FUNCTION_BLOCK "SysTime"   // FB10, SCL
TITLE = 'Формируем текущее циклическое системное время в MD20 (_TIME)'
{ S7_Optimized_Access := 'FALSE' }
AUTHOR : SAA
FAMILY : xSYSTEM
NAME : SysTime
VERSION : 4.0
// // Особенностью SFC 64 TIME_TCK является выдача времени в [мс]
// // от 0 до 16#7FFFFFFF т.е. необходимо организовать переход
// // от 0 до 16#FFFFFFFF. Побочно вычисляем текущее, максимальное
// // и минимальное время цикла и время работы в [сек]
   VAR_OUTPUT
      Tsek : DInt := 0;   // Текущее время [с]
      Tnow : Time := T#0MS;   // Текущее время цикла [мс]
      Trxm : Real := 0.0;   // Текущее время цикла [с]
      Tmid : Real := 0.0;   // Сглаженное время цикла [с]
      Tmax : Time := T#0MS;   // Максимальное время цикла [мс]
      Tmin : Time := T#24D;   // Минимальное время цикла [мс]
      DTx : Date_And_Time;   // Текущее время PLC
   END_VAR
   VAR
      Tm : Time := T#0MS;   // Сохраненное системное время
      Ts : Time := T#0MS;   // Накопитель для секундного счета
      NSc : Bool := 0;   // Первый проход выполнен
   END_VAR
   VAR_TEMP
      Tx : Time;   // Текущее системное время [мс]
      RV : Int;   // RETVAL
   END_VAR
BEGIN

   // Получаем текущее время PLC
   #RV := RD_LOC_T(OUT => #DTx);
   // Получаем разницу между вызовами TIME_TCK
   #Tx := TIME_TCK();
   #Tnow := T_CONV(INT_TO_DINT(DINT_TO_INT(T_CONV(#Tx - #Tm))));
   #Trxm := DINT_TO_REAL(T_CONV(#Tnow)) * 0.001;
   "_Time_dR" := #Trxm;
   #Tm := #Tx;
   // При перезапуске исключаем ударное изменение времени
   IF ("_ReStart") THEN
       #Tnow := T#0s;
   END_IF;
   // Увеличиваем текущий счетчик системного времени
   "_Time" := "_Time" + #Tnow;
   // Пропускаем первый цикл
   IF (#NSc) THEN
       // Выбираем максимум и минимум цикла
       IF (#NSc & #Tnow > #Tmax) THEN
           #Tmax := #Tnow;
       END_IF;
       IF (#NSc & #Tnow < #Tmin) THEN
           #Tmin := #Tnow;
       END_IF;
       // Сглаженное время цикла [с]
       #Tmid := (#Trxm - #Tmid) * 0.001 + #Tmid;
   END_IF;
   // Получаем время в секундах
   #Ts := #Ts + #Tnow;
   IF (#Ts >= T#1s) THEN
       #Tsek := #Tsek + 1;
       #Ts := #Ts - T#1s;
   END_IF;
   // Устанавливаем флаг выполнения первого прохода
   #NSc := 1;
   // Текущее системное время в "_TIME"
END_FUNCTION_BLOCK

FUNCTION_BLOCK "AiCh_My"   // FB12, SCL
{ S7_Optimized_Access := 'FALSE' }
VERSION : 0.1
   VAR_INPUT
      Yi : Int;   // Текущее значение аналогового входного канала
      Ymax : Int := 27648;   // Значение PIW/PID(Ai/Ad) при 100% входного диапазона
      Ymin : Int;   // Значение PIW/PID(Ai/Ad) при 0% входного диапазона
      Xmax : Real;   // Номинал Px при Ai=100%
      Xmin : Real;   // Номинал Px при Ai=0%
      Ke : Bool;   // Прямое использование канала
      Kf : Real;   // Коэффициент преобразования Ai=>Px (множитель)
      lag_koef : Real := 1.0;   // Множитель для сглаживания колебаний входного сигнала
      PV_AH_Lim : Real;   // Максимальний уровень сигнала
      PV_AL_Lim : Real;   // Минимальный уровень сигнала
      PV_WH_Lim : Real;   // Высокий уровень сигнала
      PV_WL_Lim : Real;   // Низкий уровень сигнала
      EnableAL_Lim : Bool := 1;
   END_VAR
   VAR_OUTPUT
      NDB : UDInt := 0;   // Номер InstanceDB
      Pz : Real;   // Фактическое значение канала
      Px : Real;   // Рабочее значение канала
      AH_LIM : Bool;
      AL_LIM : Bool;
   END_VAR
   VAR
      Alarm_error : Program_Alarm;
      Alarm_AH_Lim : Program_Alarm;
      Alarm_AL_Lim : Program_Alarm;
      Alarm_WH_Lim : Program_Alarm;
      Alarm_WL_Lim : Program_Alarm;
      ME : "DrvME";   // Набор данных для обработки ALARM_D
      initBlock : Bool;
      err : Bool;
   END_VAR
   VAR_TEMP
      Pu : Real;
      TSA : "TANY";   // Структура ANY для определения InstanceDB
      TPA AT TSA : ANY;   // Указатель ANY для определения InstanceDB
   END_VAR
BEGIN
   #err := (#Yi <= -32767 OR #Yi >= 32767);

   IF #Ymax - #Ymin <> 0 AND NOT #err THEN
       IF #Ke THEN
           #Pz := #Yi * #Kf+#Xmin;
       ELSE
           #Pz := ((INT_TO_REAL(#Yi - #Ymin)) / (INT_TO_REAL(#Ymax - #Ymin))) * (#Xmax - #Xmin) + #Xmin;
       END_IF;
      // Сглаживание сигнала
       #Pu := #Pz;
       #Pu := (#Pu - #Px) * #lag_koef + #Px;
       #Px := #Pu;

       IF #Pz < #Xmin THEN
           #Pz := #Xmin;
       END_IF;

       IF #Px < #Xmin THEN
           #Px := #Xmin;
       END_IF;

   ELSE
       IF #Yi <= -32767 THEN
           #Pz := -99.0;
           #Px := -99.0;
       END_IF;

       IF #Yi >= 32767 THEN
           #Pz := 999.0;
           #Px := 999.0;
       END_IF;

       IF #Ymax - #Ymin = 0 THEN
           #Pz := -1.0;
           #Px := -1.0;
       END_IF;
   END_IF;


   // Запрос на инициализацию данных
   IF NOT #initBlock THEN
   // Инициализация данных
       #ME.Pr.N2 := 0;
       #ME.Pr.N3 := 0;
       #ME.Pr.N4 := 0;
       #ME.Pr.N5 := 0;
       #ME.Pr.N6 := 0;
   // Устанавливаем номер данного Instance Data Block
       #TPA := #ME;
       #NDB := #TSA.PTR.DN;
       #initBlock := 1;
   END_IF;


   // Сообщение: Неисправность канала датчика
   #ME.Pr.N1 := #NDB*10;
   #ME.Pr.N4 := #NDB*10;
   #Alarm_error(SIG := #err,
                TIMESTAMP := "TS0",
                SD_1:=#ME.Pr.N1, SD_2 := #ME.Pr.N4);


   // Сообщение: Максимальний уровень
   #AH_LIM := #Px > #PV_AH_Lim AND NOT #err;
   #Alarm_AH_Lim(SIG := #AH_LIM,
                  TIMESTAMP := "TS0",
                  SD_1 := #ME.Pr.N1, SD_2 := #ME.Pr.N4);

    // // Сообщение: Минимальный уровень
    #AL_LIM := #Px < #PV_AL_Lim AND NOT #err;
    #Alarm_AL_Lim(SIG :=#AL_LIM AND #EnableAL_Lim,
                  TIMESTAMP := "TS0",
                  SD_1 := #ME.Pr.N1, SD_2 := #ME.Pr.N4);

    // Сообщение: Высокий уровень
    // #Alarm_WH_Lim(SIG := #Px > #PV_WH_Lim AND NOT #err,
    //               TIMESTAMP := "TS0",
    //               SD_1 := #ME.Pr.N1);

    // Сообщение: Низкий уровень
    // #Alarm_WL_Lim(SIG := #Px < #PV_WL_Lim AND NOT #err,
    //               TIMESTAMP := "TS0",
    //               SD_1 := #ME.Pr.N1);
END_FUNCTION_BLOCK

FUNCTION_BLOCK "FpDW"   // FB18, SCL
{ S7_Optimized_Access := 'FALSE' }
VERSION : 0.1
   VAR
      F : Array[00..95] of Bool;   // Текущее состояние
      D AT F : Array[0..2] of DWord;
      "B" : Array[0..2] of DWord;   // Сохраненное состояние
      Fx : Bool := 0;   // Наличие текущих активных сигналов
      Fp : Bool := 0;   // Импульс при наличии новых сигналов
      Fe : Bool := 0;   // Наличие не сквитированных сигналов
      Fa : Bool := 0;   // Мигающий признак Fe
      Fm : Bool := 0;   // Поиск фронта квитирования
   END_VAR
BEGIN
   // ------------------------------------------------------------------------------------------------------------------------------------------------
   // Квитирование (сброс признака наличия новых сигналов)
   IF (#Fm XOR "_ACK") THEN
       #Fe := #Fe & #Fm;
       #Fm := "_ACK";
   END_IF;
   // ------------------------------------------------------------------------------------------------------------------------------------------------
   // Проверка наличия активных сообщений
   #Fx := (#D[0] OR #D[1] OR #D[2]) <> 0;
   // Проверка наличия новых сообщений
   #Fp := ((#D[0] XOR #"B"[0]) & #D[0] OR (#D[1] XOR #"B"[1]) & #D[1] OR (#D[2] XOR #"B"[2]) & #D[2]) <> 0;
   #Fe := #Fe OR #Fp;
   #Fa := (#Fe & "_Clk08sec") OR (#Fx & NOT #Fe);
   // ------------------------------------------------------------------------------------------------------------------------------------------------
   // Сохранение состояния
   #"B" := #D;
   // Очистка входных данных на время наладки
   // #D[0] := 0;
   // #D[1] := 0;
   // #D[2] := 0;
   // ------------------------------------------------------------------------------------------------------------------------------------------------
END_FUNCTION_BLOCK

FUNCTION_BLOCK "DrvCell"   // FB20, SCL
TITLE = 'Элементарная ячейка управления механизмом (DrvCell)'
{ S7_Optimized_Access := 'FALSE' }
AUTHOR : SAA
FAMILY : xDRIVER
NAME : DrvCell
VERSION : 4.0
// ; S7_blockview := 'small'
   VAR_INPUT
      GRP : UDInt := 0;   // Группа механизмов для HMI
      Chr : DWord := 0;   // Входное слово командного канала
      CFr AT Chr : "DrvCF";
      STr AT Chr : "DrvST";
      Lnr : Bool := 1;   // Наличие связи в линии командного канала
      STu : DWord := 16#1000;   // Дополнительные флаги в слове состояния ST
      SQ1 : Bool := 0;   // Концевой выключатель для Km1
      SQ2 : Bool := 0;   // Концевой выключатель для Km2
      Kx1 : Bool := 0;   // Блок-контакт Km1 (подтверждение срабатывания Km1==Kx1)
      Kx2 : Bool := 0;   // Блок-контакт Km2 (подтверждение срабатывания Km2==Kx2)
      KxA : Bool := 0;   // Блок-контакт Km1&Km2 (совмещенный в механизме)
      KxB : Bool := 0;   // Блок-контакт байпаса (разгон окончен)
      QFx : Bool := 1;   // Питающий автомат цепей механизма (1==включен)
      Flt : Bool := 0;   // Внешняя неисправность (блокирующая) (1==активна по умолчанию)
      Dis : Bool := 0;   // Запрет работы ('Аварийный СТОП' или другой режим) (1==активен)
      Ds1 : Bool := 0;   // Блокировка включения (принудительное отключение) Km1
      Ds2 : Bool := 0;   // Блокировка включения (принудительное отключение) Km2
      DsA : Bool := 0;   // Общая блокировка включения (принудительное отключение) Km1&Km2
      MEn : Bool := 1;   // Разрешение выдачи сообщений для HMI
      Mdx : Bool := 0;   // Режим работы (0==Ручной/1==Автомат)
      Cm1 : Bool := 0;   // Включить Km1 (команда в Mode==1)
      Cm2 : Bool := 0;   // Включить Km2 (команда в Mode==1)
      SB1 : Bool := 0;   // Кнопка включения Km1 (фронт активен) (с фиксацией или без)
      SB2 : Bool := 0;   // Кнопка включения Km2 (фронт активен) (с фиксацией или без)
      OFF : Bool := 0;   // Кнопка 'СТОП' для снятия фиксации (1==активен)
      Ack : Bool := 0;   // Сброс индикации ошибки (квитирование) (1==активен)
      SBe : Bool := 1;   // Разрешение кнопок (при ==0 запрет без отключения)
      SP1 : SInt := 100;   // Уставка задания Km1 (-100..+100)[%] (режим: Ручной)
      SP2 : SInt := -100;   // Уставка задания Km2 (-100..+100)[%] (режим: Ручной)
      SK1 : SInt := 100;   // Уставка задания Km1 (-100..+100)[%] (режим: Автомат)
      SK2 : SInt := -100;   // Уставка задания Km2 (-100..+100)[%] (режим: Автомат)
      Kb_Sb1 : Bool := 0;   // Кнопка SB1 без фиксации (Km1 отключается после отпускания SB1)
      Kb_Sr1 : Bool := 0;   // Кнопка SB1 в режиме переключателя (Вкл/Откл одной кнопкой)
      Kb_Sb2 : Bool := 0;   // Кнопка SB2 без фиксации (Km2 отключается после отпускания SB2)
      Kb_Sr2 : Bool := 0;   // Кнопка SB2 в режиме переключателя (Вкл/Откл одной кнопкой)
      Kb_Ls1 : Bool := 0;   // Индикация Km1 желтым светом (Lr+Lg)
      Kb_Ls2 : Bool := 0;   // Индикация Km2 желтым светом (Lr+Lg)
      Kb_LsA : Bool := 0;   // Используется общая подсветка на оба канала Km1/Km2
      Kb_LsH : Bool := 0;   // Моноцветная импульсная индикация неисправностей
      Kb_HMI : Bool := 0;   // Кнопки в режиме импульса HMI (сброс после использования)
      Ds : DWord := 0;   // Канал системы блокировок
      Nm AT Ds : "DrvNm";
      Md_KxB : Bool := 0;   // KxB выпоняет роль блок-контакта байпаса (разгон окончен)
      Md_SQA : Bool := 0;   // Разрешено наличие обоих SQ одновременно
      Md_RsM : Bool := 0;   // Отключение Km при переходе в ручной режим (Mdx=>0)
      Md_DsE : Bool := 0;   // Разрешено аварийное отключение без выдержки времени
      Md_DsM : Bool := 0;   // Не учитывать блокировку действия как Err+Ds в Mdx==0
      Md_DsA : Bool := 0;   // Не учитывать блокировку действия как Err+Ds в Mdx==1
      Md_RsE : Bool := 0;   // Сброс счетчика отработанного времени по фронту Km1/Km2
      Md_Ack : Bool := 0;   // Сброс сообщений производить по обратному фронту Ack
      Md_Tx1 : Bool := 0;   // Используется отключение Km1 по таймеру Tm1
      Md_Sx1 : Bool := 0;   // Превышение времени работы с Sx1==0 является неисправностью
      Md_Sn1 : Bool := 0;   // Разрешен съезд с SQ1 (Sx1=>0) без команды (при On==0)
      Md_Km1 : Bool := 0;   // Активный сигнал SQ1 отключает Km1 (для удержания установить 0)
      Md_Kx1 : Bool := 0;   // Kx1 выпоняет роль блок-контакта (должен соответствовать Km1)
      Md_Tx2 : Bool := 0;   // Используется отключение Km2 по таймеру Tm2
      Md_Sx2 : Bool := 0;   // Превышение времени работы с Sx2==0 является неисправностью
      Md_Sn2 : Bool := 0;   // Разрешен съезд с SQ2 (Sx2=>0) без команды (при On==0)
      Md_Km2 : Bool := 0;   // Активный сигнал SQ2 отключает Km2 (для удержания установить 0)
      Md_Kx2 : Bool := 0;   // Kx2 выпоняет роль блок-контакта (должен соответствовать Km2)
      Md_Sxx : Bool := 0;   // Необходима проверка SQ2 после отключения Km1
      Md_Tm1 : Time := T#24D;   // Контроль времени работы Km1 (T#0MS/T#24D - без ограничения)
      Md_Tm2 : Time := T#24D;   // Контроль времени работы Km2 (T#0MS/T#24D - без ограничения)
      Md_TmX : Time := T#1S;   // Контроль времени включения Km1&Km2 по БК Kx1&Kx2&KxA
      Md_TmD : Time := T#1S;   // Контроль времени отключения Km1&Km2 по БК Kx1&Kx2&KxA
      Md_TmS : Time := T#0MS;   // Уставка времени разгона после включения KOn
      Md_TmF : Time := T#0MS;   // Уставка времени выбега после отключения KOn
      Md_TmU : Time := T#0MS;   // Уставка времени растормаживания перед пуском Km
      Md_TmL : Time := T#0MS;   // Уставка времени наложения тормоза после отключения KOn
   END_VAR
   VAR_OUTPUT
      NDB : UDInt := 0;   // Номер InstanceDB
      Chx : DWord := 0;   // Исходное слово командного канала
      CFx AT Chx : "DrvCF";
      STx AT Chx : "DrvST";
      Sx1 : Bool := 0;   // Активен SQ1 (Sx1==1)
      Sx2 : Bool := 0;   // Активен SQ2 (Sx2==1)
      Sr1 : Bool := 0;   // Механизм в положении Sx1 (рабочее) и остановлен
      Sr2 : Bool := 0;   // Механизм в положении Sx2 (исходное) и остановлен
      Ks1 : Bool := 0;   // Управление действием Km1 от SB1
      Ks2 : Bool := 0;   // Управление действием Km2 от SB2
      KGo : Bool := 0;   // Наличие активной команды Ks1&Ks2
      KBr : Bool := 0;   // Включение тормоза (растормаживание)
      Km1 : Bool := 0;   // Включен Km1 (контактор замкнут с перекрытием)
      Km2 : Bool := 0;   // Включен Km2 (контактор замкнут с перекрытием)
      KOn : Bool := 0;   // Включено (контакторы замкнуты с перекрытием)
      Run : Bool := 0;   // Разгон закончен (стабильный участок)
      Lg1 : Bool := 0;   // Индикация действия от SB1 (зеленый)
      Lg2 : Bool := 0;   // Индикация действия от SB2 (зеленый)
      Lr1 : Bool := 0;   // Индикация действия от SB1 (красный)
      Lr2 : Bool := 0;   // Индикация действия от SB2 (красный)
      Rdy : Bool := 0;   // Механизм готов к включению (нет Err)
      Err : Bool := 0;   // Общая неисправность (Err==1) необходимо квитирование
      Dsx : Bool := 0;   // Запрет работы ('Аварийный СТОП') (1==активен)
      Msx : Bool := 0;   // Запрет выдачи сообщений для HMI (групповое) (1==активен)
      Acx : Bool := 0;   // Выход квитирования (дублирование Ack)
      ST : DWord := 0;   // Состояние механизма (для HMI)
   END_VAR
   VAR_IN_OUT
      TmE : UDInt := 0;   // Прошедшее с начала отсчета рабочее время [сек]
   END_VAR
   VAR
      MsSr1 : Program_Alarm;   // Не сработал КВ SQ1 за заданное время Tm1
      MsSr2 : Program_Alarm;   // Не сработал КВ SQ2 за заданное время Tm2
      MsSe1 : Program_Alarm;   // Механизм без команды сошел с КВ SQ1
      MsSe2 : Program_Alarm;   // Механизм без команды сошел с КВ SQ2
      MsSeA : Program_Alarm;   // Одновременно активны оба КВ SQ1 и SQ2
      MsKeB : Program_Alarm;   // БК KxB не соответствует состоянию KOn
      MsKe1 : Program_Alarm;   // БК Kx1 не соответствует контактору Km1
      MsKe2 : Program_Alarm;   // БК Kx2 не соответствует контактору Km2
      MsDs1 : Program_Alarm;   // Действие Km1 заблокировано (Ds1/DsA)
      MsDs2 : Program_Alarm;   // Действие Km2 заблокировано (Ds2/DsA)
      MsQFe : Program_Alarm;   // Отключен автоматический выключатель
      MsFlt : Program_Alarm;   // Внешняя неисправность (блокирующая)
      MsErr : Program_Alarm;   // Внутренняя неисправность DrvCell
      SbM : "DrvSb";   // Локальный блок обработки кнопочных комманд
      Chm : DWord := 0;   // Хранилище входящего командного канала
      CFm AT Chm : "DrvCF";
      STm AT Chm : "DrvST";
      FSc : Bool := 1;   // Первый проход блока (необходима инициализация)
      Tm : Struct   // Хранилище флагов и данных таймеров
         Ts : Time := T#0MS;   // Сохраненное системное время
         Tw : Time := T#0MS;   // Накопительный счетчик времени TmE
         Br : Time := T#0MS;   // Контрольное время тормоза
         Km : Time := T#0MS;   // Контрольное время контакторов
         On : Time := T#0MS;   // Контрольное время пускателя
         Tm1 : Bool := 0;   // Контроль времени работы Km1 производится (Tm1<T#24D)
         Tm2 : Bool := 0;   // Контроль времени работы Km2 производится (Tm2<T#24D)
         Km1 : Bool := 0;   // Последним производилось отключение Km1
         Km2 : Bool := 0;   // Последним производилось отключение Km2
         r00 : Word := 0;   // ----
      END_STRUCT;
      BFm : DWord := 0;   // Хранилище флагов (Буффер для текущих флагов)
      Ms : "DrvMs";   // Текущие аварийные сообщения DrvCell для просмотра в VAT
      Hs AT Ms : DWord;   // Хранилище сообщений (Буффер для текущих флагов сообщений)
      MF : Struct   // Структура содержит информацию о вызовах ALARM
         Hs : "DrvMs";   // Предыдущее состояние флагов сообщений
         Md : "DrvMs";   // Маркировка событий Mdx==1 (DrvCell в автоматическом режиме)
         Rn : "DrvMs";   // Маркировка событий KGo==1 (DrvCell был включен до сообщения)
         Ms : "DrvMs";   // Маркировка событий Mse==0 (Нет разрешения сообщений для HMI)
         D1 : Word := 0;   // Дополнительная строка из таблицы DrvNm для Ds1
         D2 : Word := 0;   // Дополнительная строка из таблицы DrvNm для Ds2
      END_STRUCT;
      MU AT MF : Struct   // Структура содержит информацию о вызовах ALARM
         Hs : DWord;   // Предыдущее состояние флагов сообщений
         Md : DWord;   // Маркировка событий Mdx==1 (DrvCell в автоматическом режиме)
         Rn : DWord;   // Маркировка событий KGo==1 (DrvCell был включен до сообщения)
         Ms : DWord;   // Маркировка событий Mse==0 (Нет разрешения сообщений для HMI)
      END_STRUCT;
      ME : "DrvME";   // Набор данных для обработки ALARM
   END_VAR
   VAR_TEMP
      TSA : "TANY";   // Структура ANY для определения InstanceDB
      TPA AT TSA : ANY;   // Указатель ANY для определения InstanceDB
      Fx : Struct   // Внутренние флаги состояния
         Kx1 : Bool;   // Блок-контакт Km1 (подтверждение срабатывания Km1==Kx1)
         Kx2 : Bool;   // Блок-контакт Km2 (подтверждение срабатывания Km2==Kx2)
         KxA : Bool;   // Блок-контакт Km1&Km2 (совмещенный в механизме)
         KxB : Bool;   // Блок-контакт байпаса (разгон окончен)
         QFx : Bool;   // Питающий автомат цепей механизма (1==включен)
         Flt : Bool;   // Внешняя неисправность (блокирующая) (1==активна по умолчанию)
         Dis : Bool;   // Запрет работы ('Аварийный СТОП' или другой режим) (1==активен)
         Ds1 : Bool;   // Блокировка включения (принудительное отключение) Km1
         Ds2 : Bool;   // Блокировка включения (принудительное отключение) Km2
         Mdx : Bool;   // Рабочие режимы работы (0==Ручной/1==Автомат)
         Cm1 : Bool;   // Включить Km1 (команда в Mode==1)
         Cm2 : Bool;   // Включить Km2 (команда в Mode==1)
         Sx1 : Bool;   // Активное состояние SQ1
         Sx2 : Bool;   // Активное состояние SQ2
         Ks1 : Bool;   // Запрос на включение Km1
         Ks2 : Bool;   // Запрос на включение Km2
         KGo : Bool;   // Наличие активной команды Ks1&Ks2
         KBr : Bool;   // Включение тормоза (растормаживание)
         Km1 : Bool;   // Включен Km1 (контактор замкнут с перекрытием)
         Km2 : Bool;   // Включен Km2 (контактор замкнут с перекрытием)
         KOn : Bool;   // Включено (контакторы замкнуты с перекрытием)
         Run : Bool;   // Разгон закончен (стабильный участок)
         Err : Bool;   // Наличие не сквитированной неисправности
         r00 : Bool;   // ----
         Tm1 : Bool;   // Контроль времени работы Km1 (T#0MS/T#24D - без ограничения)
         Tm2 : Bool;   // Контроль времени работы Km2 (T#0MS/T#24D - без ограничения)
         TmX : Bool;   // Контроль времени включения Km1&Km2 по БК Kx1&Kx2&KxA
         TmD : Bool;   // Контроль времени отключения Km1&Km2 по БК Kx1&Kx2&KxA
         TmS : Bool;   // Уставка времени разгона после включения KOn
         TmF : Bool;   // Уставка времени выбега после отключения KOn
         TmU : Bool;   // Уставка времени растормаживания перед пуском Km
         TmL : Bool;   // Уставка времени наложения тормоза после отключения KOn
      END_STRUCT;
      Dx AT Fx : DWord;   // Буффер для текущих флагов
      Fm : Struct   // Внутренние флаги состояния
         Kx1 : Bool;   // Блок-контакт Km1 (подтверждение срабатывания Km1==Kx1)
         Kx2 : Bool;   // Блок-контакт Km2 (подтверждение срабатывания Km2==Kx2)
         KxA : Bool;   // Блок-контакт Km1&Km2 (совмещенный в механизме)
         KxB : Bool;   // Блок-контакт байпаса (разгон окончен)
         QFx : Bool;   // Питающий автомат цепей механизма (1==включен)
         Flt : Bool;   // Внешняя неисправность (блокирующая) (1==активна по умолчанию)
         Dis : Bool;   // Запрет работы ('Аварийный СТОП' или другой режим) (1==активен)
         Ds1 : Bool;   // Блокировка включения (принудительное отключение) Km1
         Ds2 : Bool;   // Блокировка включения (принудительное отключение) Km2
         Mdx : Bool;   // Рабочие режимы работы (0==Ручной/1==Автомат)
         Cm1 : Bool;   // Включить Km1 (команда в Mode==1)
         Cm2 : Bool;   // Включить Km2 (команда в Mode==1)
         Sx1 : Bool;   // Активное состояние SQ1
         Sx2 : Bool;   // Активное состояние SQ2
         Ks1 : Bool;   // Запрос на включение Km1
         Ks2 : Bool;   // Запрос на включение Km2
         KGo : Bool;   // Наличие активной команды Ks1&Ks2
         KBr : Bool;   // Включение тормоза (растормаживание)
         Km1 : Bool;   // Включен Km1 (контактор замкнут с перекрытием)
         Km2 : Bool;   // Включен Km2 (контактор замкнут с перекрытием)
         KOn : Bool;   // Включено (контакторы замкнуты с перекрытием)
         Run : Bool;   // Разгон закончен (стабильный участок)
         Err : Bool;   // Наличие не сквитированной неисправности
         r00 : Bool;   // ----
         Tm1 : Bool;   // Контроль времени работы Km1 (T#0MS/T#24D - без ограничения)
         Tm2 : Bool;   // Контроль времени работы Km2 (T#0MS/T#24D - без ограничения)
         TmX : Bool;   // Контроль времени включения Km1&Km2 по БК Kx1&Kx2&KxA
         TmD : Bool;   // Контроль времени отключения Km1&Km2 по БК Kx1&Kx2&KxA
         TmS : Bool;   // Уставка времени разгона после включения KOn
         TmF : Bool;   // Уставка времени выбега после отключения KOn
         TmU : Bool;   // Уставка времени растормаживания перед пуском Km
         TmL : Bool;   // Уставка времени наложения тормоза после отключения KOn
      END_STRUCT;
      Dm AT Fm : DWord;   // Буффер для сохраненных флагов
      Fp : Struct   // Внутренние флаги состояния
         Kx1 : Bool;   // Блок-контакт Km1 (подтверждение срабатывания Km1==Kx1)
         Kx2 : Bool;   // Блок-контакт Km2 (подтверждение срабатывания Km2==Kx2)
         KxA : Bool;   // Блок-контакт Km1&Km2 (совмещенный в механизме)
         KxB : Bool;   // Блок-контакт байпаса (разгон окончен)
         QFx : Bool;   // Питающий автомат цепей механизма (1==включен)
         Flt : Bool;   // Внешняя неисправность (блокирующая) (1==активна по умолчанию)
         Dis : Bool;   // Запрет работы ('Аварийный СТОП' или другой режим) (1==активен)
         Ds1 : Bool;   // Блокировка включения (принудительное отключение) Km1
         Ds2 : Bool;   // Блокировка включения (принудительное отключение) Km2
         Mdx : Bool;   // Рабочие режимы работы (0==Ручной/1==Автомат)
         Cm1 : Bool;   // Включить Km1 (команда в Mode==1)
         Cm2 : Bool;   // Включить Km2 (команда в Mode==1)
         Sx1 : Bool;   // Активное состояние SQ1
         Sx2 : Bool;   // Активное состояние SQ2
         Ks1 : Bool;   // Запрос на включение Km1
         Ks2 : Bool;   // Запрос на включение Km2
         KGo : Bool;   // Наличие активной команды Ks1&Ks2
         KBr : Bool;   // Включение тормоза (растормаживание)
         Km1 : Bool;   // Включен Km1 (контактор замкнут с перекрытием)
         Km2 : Bool;   // Включен Km2 (контактор замкнут с перекрытием)
         KOn : Bool;   // Включено (контакторы замкнуты с перекрытием)
         Run : Bool;   // Разгон закончен (стабильный участок)
         Err : Bool;   // Наличие не сквитированной неисправности
         r00 : Bool;   // ----
         Tm1 : Bool;   // Контроль времени работы Km1 (T#0MS/T#24D - без ограничения)
         Tm2 : Bool;   // Контроль времени работы Km2 (T#0MS/T#24D - без ограничения)
         TmX : Bool;   // Контроль времени включения Km1&Km2 по БК Kx1&Kx2&KxA
         TmD : Bool;   // Контроль времени отключения Km1&Km2 по БК Kx1&Kx2&KxA
         TmS : Bool;   // Уставка времени разгона после включения KOn
         TmF : Bool;   // Уставка времени выбега после отключения KOn
         TmU : Bool;   // Уставка времени растормаживания перед пуском Km
         TmL : Bool;   // Уставка времени наложения тормоза после отключения KOn
      END_STRUCT;
      Dp AT Fp : DWord;   // Буффер для признаков изменения флагов
      Mx : "DrvMs";   // Текущие аварийные сообщения DrvCell для HMI
      Hx AT Mx : DWord;   // Буффер для сохраненных флагов сообщений
      Mp : "DrvMs";   // Текущие аварийные сообщения DrvCell для HMI
      Hp AT Mp : DWord;   // Буффер для сохраненных флагов сообщений
      Chk : DWord;   // Хранилище (временное) командного канала
      CFk AT Chk : "DrvCF";
      STk AT Chk : "DrvST";
      Fk : Struct   // Обработка сигналов канала управления
         SB1 : Bool;   // Команда SA1/SB1 на включение Km1
         SB2 : Bool;   // Команда SA2/SB2 на включение Km2
         OFF : Bool;   // Команда OFF на отключение Km1 и Km2
         CmA : Bool;   // Текущая команда активна
         EvN : Bool;   // Зафиксирована новая команда
      END_STRUCT;
      Fw AT Fk : Word;
      CmB : Struct   // Быстрое преобразование BYTE2WORD
         H : Byte;
         L : Byte;
      END_STRUCT;
      CmW AT CmB : Word;
      Fe : Bool;   // Флаг отсутствия аварийного отключения
      Mz : Bool;   // Флаг разрешения сообщений ALARM
      Fa : Bool;   // Временные промежуточные флаги
      F0 : Bool;   // Временные промежуточные флаги
      F1 : Bool;   // Временные промежуточные флаги
      F2 : Bool;   // Временные промежуточные флаги
   END_VAR
   VAR CONSTANT
      MkErr : DWord := DW#16#FFFF0000;   // Маска флагов сообщений в слове статуса
      MkErA : DWord := DW#16#1CF00000;   // Маска флагов сообщений квитируемых с проверкой
      MkErM : DWord := DW#16#0000FFFF;   // Маска квитирования флагов сообщений
   END_VAR
BEGIN
   // Сброс флагов команд
   #Fw := 0;

   // Первичное событие при инициализации
   #Fa := #FSc;
   // Запрос на инициализацию данных
   IF (#FSc) THEN
       // Инициализация данных
       #ME.Pr.N2 := 0;
       #ME.Pr.N4 := 0;
       #ME.Pr.N5 := 0;
       // Устанавливаем номер данного Instance Data Block
       #TPA := #ME;
       #NDB := #TSA.PTR.DN;
       // Назначаем группу сообщений (механизмов)
       IF (#GRP = 0) THEN
           #GRP := #NDB * 100;
       END_IF;
       // Сбрасываем флаг первого цикла
       #FSc := 0;
   END_IF;
   // Вызов блока обработки кнопок с актуальным STx
   #SbM.Drv := 1;
   #STr.STx := #STx.STx;
   #SbM(Chr := #Chr,
        Lnr := #Lnr,
        SB1 := #SB1,
        SB2 := #SB2,
        OFF := #OFF,
        Ack := #Ack,
        SBe := #SBe,
        SP1 := #SP1,
        SP2 := #SP2,
        Kb_Sb1 := #Kb_Sb1,
        Kb_Sr1 := #Kb_Sr1,
        Kb_Sb2 := #Kb_Sb2,
        Kb_Sr2 := #Kb_Sr2,
        Kb_Ls1 := #Kb_Ls1,
        Kb_Ls2 := #Kb_Ls2,
        Kb_LsA := #Kb_LsA,
        Kb_LsH := #Kb_LsH,
        Kb_HMI := #Kb_HMI,
        Lg1 => #Lg1,
        Lg2 => #Lg2,
        Lr1 => #Lr1,
        Lr2 => #Lr2);
   // Сохраняем состояние кнопок
   #SB1 := #SbM.SB1;
   #SB2 := #SbM.SB2;
   #OFF := #SbM.OFF;
   #Ack := #SbM.Ack;
   // Сохраняем индикацию для HMI
   #Ms.Lg1 := #Lg1 & NOT #Lr1;
   #Ms.Lg2 := #Lg2 & NOT #Lr2;
   #Ms.Lr1 := #Lr1 & NOT #Lg1;
   #Ms.Lr2 := #Lr2 & NOT #Lg2;
   #Ms.Ly1 := #Lg1 & #Lr1;
   #Ms.Ly2 := #Lg2 & #Lr2;

   // Загружаем текущие флаги состояния DrvCell
   #Dm := #BFm;
   #Dx := #BFm;
   #Fx.Sx1 := #SQ1;// Активное состояние SQ1
   #Fx.Sx2 := #SQ2;// Активное состояние SQ2
   #Fx.Kx1 := #Kx1;// Блок-контакт Km1 (подтверждение срабатывания Km1==Kx1)
   #Fx.Kx2 := #Kx2;// Блок-контакт Km2 (подтверждение срабатывания Km2==Kx2)
   #Fx.KxA := #KxA;// Блок-контакт Km1&Km2 (совмещенный в механизме)
   #Fx.KxB := #KxB;// Блок-контакт байпаса (разгон окончен)
   #Fx.QFx := #QFx;// Питающий автомат цепей механизма (1==включен)
   #Fx.Flt := #Flt;// Внешняя неисправность (блокирующая) (1==активна по умолчанию)
   #Fx.Dis := #Dis OR "_HALT";// Запрет работы ('Аварийный СТОП' или другой режим)  (1==активен)
   #Fx.Ds1 := #Ds1 OR #DsA OR #Nm.Ds1 OR #Nm.DsA;// Блокировка включения (принудительное отключение) Km1
   #Fx.Ds2 := #Ds2 OR #DsA OR #Nm.Ds2 OR #Nm.DsA;// Блокировка включения (принудительное отключение) Km2
   #Fx.Mdx := #Mdx;// Рабочие режимы работы (0==Ручной/1==Автомат)
   #Fx.Cm1 := #Cm1;// Включить Km1 (команда в Mode==1)
   #Fx.Cm2 := #Cm2;// Включить Km2 (команда в Mode==1)

   // Проверяем разрешение на выдачу сообщений
   #Mz := #MEn;

   // Обрабатываем счетчик рабочего времени TmE
   IF (#Fx.Km1 OR #Fx.Km2) THEN
       #Tm.Tw := #Tm.Tw + ("_Time" - #Tm.Ts);
       IF (#Tm.Tw >= T#1s) THEN
           #Tm.Tw := #Tm.Tw - T#1s;
           #TmE := #TmE + 1;
       END_IF;
   END_IF;
   #Tm.Ts := "_Time";
   // Обрабатываем текущие таймеры Tm1&Tm2
   IF (#Fx.Tm1 & #Tm.Tm1 OR #Fx.Tm2 & #Tm.Tm2) THEN
       #Fx.Tm1 := ("_Time" - #Tm.Km < #Md_Tm1) & #Fx.Tm1;
       #Fx.Tm2 := ("_Time" - #Tm.Km < #Md_Tm2) & #Fx.Tm2;
   END_IF;
   // Обрабатываем текущие таймеры TmX&TmD
   IF (#Fx.TmX OR #Fx.TmD) THEN
       #Fx.TmX := ("_Time" - #Tm.Km < #Md_TmX) & #Fx.TmX;
       #Fx.TmD := ("_Time" - #Tm.Km < #Md_TmD) & #Fx.TmD;
   END_IF;
   // Обрабатываем текущие таймеры TmS&TmF
   IF (#Fx.TmS OR #Fx.TmF) THEN
       #Fx.TmS := ("_Time" - #Tm.On < #Md_TmS) & #Fx.TmS;
       #Fx.TmF := ("_Time" - #Tm.On < #Md_TmF) & #Fx.TmF;
   END_IF;
   // Обрабатываем текущие таймеры TmU&TmL
   IF (#Fx.TmU OR #Fx.TmL) THEN
       #Fx.TmU := ("_Time" - #Tm.Br < #Md_TmU) & #Fx.TmU;
       #Fx.TmL := ("_Time" - #Tm.Br < #Md_TmL) & #Fx.TmL;
   END_IF;

   // Устанавливаем признак наличия событий
   #Fa := #Fa OR (#Dx <> #Dm);

   // Фиксируем изменения командного канала
   #Chk := #SbM.Chx;
   IF (#Fx.Mdx = 0 & (#STk.Cmd <> #STm.Cmd)) THEN
       // Произошло событие в командном канале
       #Fa := 1;
       // Фиксируем наличие активной команды
       #Fk.CmA := #CFk.Cm2 = 0 & #CFk.Cm0 OR #CFk.Cm1;
       // Проверка получения новой команды
       #CmB.H := #STk.Cmd;
       #CmB.L := #STk.Cmd XOR #STm.Cmd;
       #Fk.EvN := NOT (((#CmW & 16#06FF) = 16#0402) OR ((#CmW & 16#07FF) = 16#0001));
       // Выделяем тип события
       #F0 := #CFk.Cm2 OR #CFk.Cm1;
       #Fk.SB1 := #F0 & #CFk.Cm0 = 0;
       #Fk.SB2 := #F0 & #CFk.Cm0 = 1;
       #Fk.OFF := #F0 = 0;
   END_IF;
   // Сохраняем текущее состояние входного командного канала
   #Chm := #SbM.Chx;

   // Результирующий сигнал квитирования
   #F0 := #CFm.Ack OR "_ACK";
   // Квитируем неисправности
   IF ((#F0 XOR #Acx) & (#F0 XOR #Md_Ack)) THEN
       // Сообщения требующие контроля KeB/Ke1/Ke2/SeA/QFe/Flt/Err
       #Fa := 1;//#Fa OR (#Hs & #MkErA) <> 0;
       // Сбрасываем активные сообщения (сохраняем статусные флаги)
       #Hs := #Hs & #MkErM;
       // Сбрасываем флаг наличия аварийных сообщений
       #Fx.Err := 0;
       #Fm.Err := 0;
       #Err := 0;
   END_IF;
   #Acx := #F0;

   // При наличии событий производим обработку тела блока DrvCell
   IF (#Fa) THEN

       // Получаем флаги событий
       #Dp := #Dx XOR #Dm;
       // Сбрасываем флаги текущих сообщений
       #Hx := 0;

       // Проверка активности и изменения SQ1
       #Mx.Sr1 := #Md_Sx1 & #Fx.Km1 & NOT (#Fx.Tm1 OR #Fx.Sx1);
       #Mx.Se1 := #Fm.Sx1 & #Fp.Sx1 & NOT (#Fx.KGo OR #Md_Sn1);
       // Проверка активности и изменения SQ2
       #Mx.Sr2 := #Md_Sx2 & #Fx.Km2 & NOT (#Fx.Tm2 OR #Fx.Sx2) OR
       #Md_Sxx & NOT (#Fx.Km1 OR #Fx.Tm2 OR #Fx.Sx2);
       #Mx.Se2 := #Fm.Sx2 & #Fp.Sx2 & NOT (#Fx.KGo OR #Md_Sn2);
       // Проверка совместной активности SQ1 и SQ2
       #Mx.SeA := #Fx.Sx1 & #Fx.Sx2 & #Md_SQA = 0;

       // Проверка блок-контактов Kx1&Kx2&KxA
       #F0 := #Fx.Kx1 & #Fx.Kx2;
       #Fa := NOT (#Fx.TmX OR #Fx.TmD);// Время перехода Вкл<->Откл истекло
       #Mx.Ke1 := #Md_Kx1 & (#F0 OR #Fa & (#Fx.Km1 XOR (#Fx.Kx1 OR #Fx.KxA & #Fx.Km2 = 0)));
       #Mx.Ke2 := #Md_Kx2 & (#F0 OR #Fa & (#Fx.Km2 XOR (#Fx.Kx2 OR #Fx.KxA & #Fx.Km1 = 0)));
       // Проверка блок-контакта KxB
       #Mx.KeB := #Md_KxB & (#Fx.KOn XOR #Fx.KxB) & (#Fx.TmS OR #Fx.TmF) = 0;

       // Обработка общих сообщений о неисправностях
       #Mx.QFe := #Fx.QFx = 0;
       #Mx.Flt := #Fx.Flt;
       #Mx.Err := #Fx.Km1 & #Fx.Km2 OR #Fx.Ks1 & #Fx.Ks2;
       #Hx := #Hx OR #Hs;
       #Fx.Err := (#Hx & #MkErr) <> 0;

       // Отключение контакторов по выдержке времени
       #Fx.Ks1 := #Fx.Ks1 & NOT (#Md_Tx1 & #Fx.Km1 & #Fx.Tm1 = 0);
       #Fx.Ks2 := #Fx.Ks2 & NOT (#Md_Tx2 & #Fx.Km2 & #Fx.Tm2 = 0);

       // Откл. Ks1 при переходе Mdx=>0
       #Fx.Ks1 := #Fx.Ks1 & NOT (#Md_RsM & #Fp.Mdx & #Fx.Mdx = 0);
       // Вкл. Ks1 по кнопке SB1 или команде Cm1
       #Fx.Ks1 := #Fx.Ks1 OR
       // В ручном режиме включаем по фронту SB1
       #Fx.Mdx = 0 & (#Fk.SB1 & #Fk.EvN) OR
       // В автомате включаем по фронту Cm1&Mdx
       #Fx.Mdx = 1 & #Fx.Cm1 & (#Fp.Mdx OR #Fp.Cm1);
       // Откл. Ks1
       IF (#Fx.Ks1) THEN
           #Fx.Ks1 := #Fx.Ks1 & NOT (
           // В ручном режиме отключаем если канал не SB1
           #Fx.Mdx = 0 & (#Fk.SB1 = 0 & (#Fk.CmA OR #Fk.EvN)) OR
           // В автомате отключаем если нет одиночной Cm1
           #Fx.Mdx = 1 & (#Fx.Cm1 = 0 OR #Fx.Cm2) OR
           // Отключение при наезде на КВ
           #Fx.Sx1 & #Md_Km1 OR
           // Отключение по сигналу СТОП
           #Fx.Dis OR
           // Отключение при неисправности
           #Fx.Err);
       END_IF;
       // Отключение при блокировке с подготовкой выдачи сообщения
       #F1 := #Fx.Ks1 & #Fx.Ds1;
       #Fx.Ks1 := #Fx.Ks1 & #F1 = 0;

       // Откл. Ks2 при переходе Mdx=>0
       #Fx.Ks2 := #Fx.Ks2 & NOT (#Md_RsM & #Fp.Mdx & #Fx.Mdx = 0);
       // Вкл. Ks2 по кнопке SB2 или команде Cm2
       #Fx.Ks2 := #Fx.Ks2 OR
       // В ручном режиме включаем по фронту SB1
       #Fx.Mdx = 0 & (#Fk.SB2 & #Fk.EvN) OR
       // В автомате включаем по фронту Cm1&Mdx
       #Fx.Mdx = 1 & #Fx.Cm2 & (#Fp.Mdx OR #Fp.Cm2);
       // Откл. Ks2
       IF (#Fx.Ks2) THEN
           #Fx.Ks2 := #Fx.Ks2 & NOT (
           // В ручном режиме отключаем если канал не SB1
           #Fx.Mdx = 0 & (#Fk.SB2 = 0 & (#Fk.CmA OR #Fk.EvN)) OR
           // В автомате отключаем если нет одиночной Cm1
           #Fx.Mdx = 1 & (#Fx.Cm2 = 0 OR #Fx.Cm1) OR
           // Отключение при наезде на КВ
           #Fx.Sx2 & #Md_Km2 OR
           // Отключение по сигналу СТОП
           #Fx.Dis OR
           // Отключение при неисправности
           #Fx.Err);
       END_IF;
       // Отключение при блокировке с подготовкой выдачи сообщения
       #F2 := #Fx.Ks2 & #Fx.Ds2;
       #Fx.Ks2 := #Fx.Ks2 & #F2 = 0;

       // Выдача сообщения при отключении блокировкой
       #Fa := #Fx.Mdx = 1 & #Md_DsA = 0 OR #Fx.Mdx = 0 & #Md_DsM = 0;
       #Mx.Ds1 := #Mx.Ds1 OR #Fa & #F1;
       #Mx.Ds2 := #Mx.Ds2 OR #Fa & #F2;
       #Fx.Err := #Fx.Err OR #Mx.Ds1 OR #Mx.Ds2;

       // Флаг отсутствия аварийного отключения и контроль таймеров
       #Fe := NOT (#Md_DsE & #Fx.Err);

       // Формирование флага наличия активной команды (KGo)
       #Fx.KGo := #Fx.Ks1 OR #Fx.Ks2;
       // Контроль времени включения тормоза (KBr)
       IF (#Fx.KGo XOR #Fm.KGo) THEN
           #Tm.Br := "_Time";
           #Fx.TmU := (#Md_TmU > T#0s) & #Fx.KGo & #Fm.KBr = 0;
           #Fx.TmL := (#Md_TmL > T#0s) & #Fm.KGo;
       END_IF;
       // Аварийный сброс таймера наложения тормоза
       #Fx.TmL := #Fx.TmL & #Fe;
       // Формирование команды включения тормоза (KBr)
       #Fx.KBr := #Fx.KGo OR #Fx.TmL;

       // Контроль времени отключения пускателя (KOn)
       IF (#Fx.KOn & NOT (#Fx.Km1 & #Fx.Ks1 OR #Fx.Km2 & #Fx.Ks2)) THEN
           #Tm.On := "_Time";
           #Fm.KOn := 0;
           #Fx.TmS := 0;
           #Fx.TmF := #Md_TmF > T#0s;
       END_IF;
       // Аварийный сброс таймера выбега пускателя
       #Fx.TmF := #Fx.TmF & #Fe;

       // Контроль условия отключения контакторов (Km1&Km2)
       #Fx.Km1 := #Fx.Km1 & #Fe & (#Fx.Ks1 OR #Fx.TmF);
       #Fx.Km2 := #Fx.Km2 & #Fe & (#Fx.Ks2 OR #Fx.TmF);
       // Контроль времени отключения контакторов (Km1&Km2)
       IF (#Fx.Km1 = 0 & #Fm.Km1 OR #Fx.Km2 = 0 & #Fm.Km2) THEN
           #Tm.Km := "_Time";
           #Fx.TmD := #Md_TmD > T#0s;
           #Fx.TmX := 0;
           #Fx.Tm1 := 0;
           #Fx.Tm2 := (#Md_Tm2 > T#0s) & #Fm.Km1 & #Md_Sxx;
           #Tm.Km1 := #Fm.Km1;
           #Tm.Km2 := #Fm.Km2;
       END_IF;
       // Аварийный сброс таймера отключения контакторов
       #Fx.TmD := #Fx.TmD & #Fe;
       // Контроль условия включения контакторов (Km1&Km2)
       #Fx.Km1 := #Fx.Km1 OR #Fx.Ks1 & NOT (#Fx.TmU OR #Fx.Kx2 OR #Fx.Km2 OR #Tm.Km1 = 0 & (#Fx.TmD OR #Fx.KxA));
       #Fx.Km2 := #Fx.Km2 OR #Fx.Ks2 & NOT (#Fx.TmU OR #Fx.Kx1 OR #Fx.Km1 OR #Tm.Km2 = 0 & (#Fx.TmD OR #Fx.KxA));
       // Контроль времени включения контакторов (Km1&Km2)
       IF (#Fm.Km1 = 0 & #Fx.Km1 OR #Fm.Km2 = 0 & #Fx.Km2) THEN
           #Tm.Km := "_Time";
           #Fx.TmX := #Md_TmX > T#0s;
           #Fx.TmD := 0;
           #Fx.Tm1 := (#Md_Tm1 > T#0s) & #Fx.Km1;
           #Fx.Tm2 := (#Md_Tm2 > T#0s) & #Fx.Km2;
           #Tm.Tm1 := #Md_Tm1 < T#24D;
           #Tm.Tm2 := #Md_Tm2 < T#24D;
           // Обработка условия сброса счетчика рабочего времени
           IF (#Md_RsE) THEN
               #TmE := 0;
               #Tm.Tw := T#0s;
           END_IF;
       END_IF;
       // Аварийный сброс таймера включения контакторов
       #Fx.TmX := #Fx.TmX & #Fe;

       // Контроль условия включения пускателя (KOn)
       #Fx.KOn := (#Fx.Ks1 & #Fx.Km1 OR #Fx.Ks2 & #Fx.Km2) & #Fx.TmX = 0;
       // Контроль времени включения пускателя (KOn)
       IF (#Fx.KOn & #Fm.KOn = 0) THEN
           #Tm.On := "_Time";
           #Fx.TmF := 0;
           #Fx.TmS := #Md_TmS > T#0s;
       END_IF;
       // Аварийный сброс таймера разгона пускателя
       #Fx.TmS := #Fx.TmS & #Fe;
       // Контроль условия флага устоявшегося режима (Run)
       #Fx.Run := #Fx.KOn & #Fx.TmS = 0;

       // Заполняем список признаков состояния сообщений DrvCell
       #Hp := (#Hs XOR #Hx) & #Hx & #MkErr;
       IF (#Hp <> 0) THEN
           // Фиксируем состояние Mdx для индикации режима
           IF (#Fx.Mdx) THEN
               #MU.Md := #MU.Md OR #Hp;
           ELSE
               #MU.Md := #MU.Md & NOT (#Hp);
           END_IF;
           // Фиксируем состояние KGo для индикации режима
           IF (#Fm.KGo) THEN
               #MU.Rn := #MU.Rn OR #Hp;
           ELSE
               #MU.Rn := #MU.Rn & NOT (#Hp);
           END_IF;
           // Фиксируем блокировку Km1
           IF (#Mp.Ds1) THEN
               IF (#Nm.DsA) THEN
                   #MF.D1 := #Nm.MsA + 75;
               ELSE
                   #MF.D1 := #Nm.Ms1 + 25;
               END_IF;
           END_IF;
           // Фиксируем блокировку Km2
           IF (#Mp.Ds2) THEN
               IF (#Nm.DsA) THEN
                   #MF.D2 := #Nm.MsA + 75;
               ELSE
                   #MF.D2 := #Nm.Ms2 + 50;
               END_IF;
           END_IF;
       END_IF;

       // Выдаем текущее состояние DrvCell на выходы
       #Sx1 := #Fx.Sx1;// Активное состояние SQ1
       #Sx2 := #Fx.Sx2;// Активное состояние SQ2
       #Ks1 := #Fx.Ks1;// Запрос на включение Km1
       #Ks2 := #Fx.Ks2;// Запрос на включение Km2
       #KGo := #Fx.KGo;// Наличие активной команды Ks1&Ks2
       #KBr := #Fx.KBr;// Включение тормоза (растормаживание)
       #Km1 := #Fx.Km1;// Включен Km1 (контактор замкнут с перекрытием)
       #Km2 := #Fx.Km2;// Включен Km2 (контактор замкнут с перекрытием)
       #KOn := #Fx.KOn;// Включено (контакторы замкнуты с перекрытием)
       #Run := #Fx.Run;// Разгон закончен (стабильный участок)
       #Err := #Fx.Err;// Наличие не сквитированной неисправности
       // Флаги организации блокировок
       #Rdy := #Fx.Err = 0;
       #Sr1 := #Fx.Sx1 & NOT (#Fx.Sx2 OR #Fx.KGo);
       #Sr2 := #Fx.Sx2 & NOT (#Fx.Sx1 OR #Fx.KGo);
       // Сохраняем текущее значение флагов
       #BFm := #Dx;

       // Сохраняем текущее значение сообщений
       #Mx.Mdx := #Fx.Mdx;// Режим работы DrvCell
       #Mx.Sx1 := #Fx.Sx1;// Активное состояние SQ1
       #Mx.Sx2 := #Fx.Sx2;// Активное состояние SQ2
       #Mx.Ks1 := #Fx.Ks1;// Запрос на включение Km1
       #Mx.Ks2 := #Fx.Ks2;// Запрос на включение Km2
       #Mx.Tm1 := #Fx.Km1 & #Fx.Tm1 = 0;// Время Tm1 истекло
       #Mx.Tm2 := #Fx.Km2 & #Fx.Tm2 = 0;// Время Tm2 истекло
       // Общая неисправность
       #F0 := #Mx.SeA OR #Mx.KeB OR #Mx.QFe OR #Mx.Flt;
       // Неисправность канала Km1
       #Mx.Er1 := #Mx.Sr1 OR #Mx.Se1 OR #Mx.Ke1 OR #Mx.Ds1 OR #F0;
       // Неисправность канала Km2
       #Mx.Er2 := #Mx.Sr2 OR #Mx.Se2 OR #Mx.Ke2 OR #Mx.Ds2 OR #F0;
       // Сохраняем флаги сообщений и статуса
       #Hs := #Hx;
       // Все события обработаны
   END_IF;

   // Заполняем список вызовов ALARM
   IF (#Mz) THEN
       // Передаются активные не обработанные сообщения
       #Hx := #Hs;
   ELSE
       // При запрете сообщений снимаем флаги передачи
       #Hx := 0;
   END_IF;
   // Генерируем передачу не обработанных аварийных сообщений
   #Hp := (#MU.Hs XOR #Hx) & #MkErr;
   IF (#Hp <> 0) THEN
       #ME.Pr.N1 := #GRP;
       // Не сработал КВ SQ1 за заданное время Tm1
       IF (#Mp.Sr1) THEN
           // Сохраняем флаги исполнения
           #ME.Pr.N2.%X2 := #MF.Md.Sr1;
           #ME.Pr.N2.%X1 := #MF.Rn.Sr1;
           #ME.Pr.N2.%X0 := #MF.Ms.Sr1;
           #ME.Pr.N6 := #GRP + 2;
           // Вызываем ALARM для активных изменений
           #MsSr1(SIG := #Mx.Sr1,
                  TIMESTAMP := "TS0",
                  SD_1 := #ME.Pr.N1,
                  SD_2 := #ME.Pr.N2,
                  SD_6 := #ME.Pr.N6);
       END_IF;
       // Не сработал КВ SQ2 за заданное время Tm2
       IF (#Mp.Sr2) THEN
           // Сохраняем флаги исполнения
           #ME.Pr.N2.%X2 := #MF.Md.Sr2;
           #ME.Pr.N2.%X1 := #MF.Rn.Sr2;
           #ME.Pr.N2.%X0 := #MF.Ms.Sr2;
           #ME.Pr.N6 := #GRP + 3;
           // Вызываем ALARM для активных изменений
           #MsSr2(SIG := #Mx.Sr2,
                  TIMESTAMP := "TS0",
                  SD_1 := #ME.Pr.N1,
                  SD_2 := #ME.Pr.N2,
                  SD_6 := #ME.Pr.N6);
       END_IF;
       // Механизм без команды сошел с КВ SQ1
       IF (#Mp.Se1) THEN
           // Сохраняем флаги исполнения
           #ME.Pr.N2.%X2 := #MF.Md.Se1;
           #ME.Pr.N2.%X1 := #MF.Rn.Se1;
           #ME.Pr.N2.%X0 := #MF.Ms.Se1;
           #ME.Pr.N6 := #GRP + 4;
           // Вызываем ALARM для активных изменений
           #MsSe1(SIG := #Mx.Se1,
                  TIMESTAMP := "TS0",
                  SD_1 := #ME.Pr.N1,
                  SD_2 := #ME.Pr.N2,
                  SD_6 := #ME.Pr.N6);
       END_IF;
       // Механизм без команды сошел с КВ SQ2
       IF (#Mp.Se2) THEN
           // Сохраняем флаги исполнения
           #ME.Pr.N2.%X2 := #MF.Md.Se2;
           #ME.Pr.N2.%X1 := #MF.Rn.Se2;
           #ME.Pr.N2.%X0 := #MF.Ms.Se2;
           #ME.Pr.N6 := #GRP + 5;
           // Вызываем ALARM для активных изменений
           #MsSe2(SIG := #Mx.Se2,
                  TIMESTAMP := "TS0",
                  SD_1 := #ME.Pr.N1,
                  SD_2 := #ME.Pr.N2,
                  SD_6 := #ME.Pr.N6);
       END_IF;
       // Одновременно активны оба КВ SQ1 и SQ2
       IF (#Mp.SeA) THEN
           // Сохраняем флаги исполнения
           #ME.Pr.N2.%X2 := #MF.Md.SeA;
           #ME.Pr.N2.%X1 := #MF.Rn.SeA;
           #ME.Pr.N2.%X0 := #MF.Ms.SeA;
           #ME.Pr.N6 := #GRP + 6;
           // Вызываем ALARM для активных изменений
           #MsSeA(SIG := #Mx.SeA,
                  TIMESTAMP := "TS0",
                  SD_1 := #ME.Pr.N1,
                  SD_2 := #ME.Pr.N2,
                  SD_6 := #ME.Pr.N6);
       END_IF;
       // БК KxB не соответствует состоянию KOn
       IF (#Mp.KeB) THEN
           // Сохраняем флаги исполнения
           #ME.Pr.N2.%X2 := #MF.Md.KeB;
           #ME.Pr.N2.%X1 := #MF.Rn.KeB;
           #ME.Pr.N2.%X0 := #MF.Ms.KeB;
           #ME.Pr.N6 := #GRP + 7;
           // Вызываем ALARM для активных изменений
           #MsKeB(SIG := #Mx.KeB,
                  TIMESTAMP := "TS0",
                  SD_1 := #ME.Pr.N1,
                  SD_2 := #ME.Pr.N2,
                  SD_6 := #ME.Pr.N6);
       END_IF;
       // БК Kx1 не соответствует контактору Km1
       IF (#Mp.Ke1) THEN
           // Сохраняем флаги исполнения
           #ME.Pr.N2.%X2 := #MF.Md.Ke1;
           #ME.Pr.N2.%X1 := #MF.Rn.Ke1;
           #ME.Pr.N2.%X0 := #MF.Ms.Ke1;
           #ME.Pr.N6 := #GRP + 8;
           // Вызываем ALARM для активных изменений
           #MsKe1(SIG := #Mx.Ke1,
                  TIMESTAMP := "TS0",
                  SD_1 := #ME.Pr.N1,
                  SD_2 := #ME.Pr.N2,
                  SD_6 := #ME.Pr.N6);
       END_IF;
       // БК Kx2 не соответствует контактору Km2
       IF (#Mp.Ke2) THEN
           // Сохраняем флаги исполнения
           #ME.Pr.N2.%X2 := #MF.Md.Ke2;
           #ME.Pr.N2.%X1 := #MF.Rn.Ke2;
           #ME.Pr.N2.%X0 := #MF.Ms.Ke2;
           #ME.Pr.N6 := #GRP + 9;
           // Вызываем ALARM для активных изменений
           #MsKe2(SIG := #Mx.Ke2,
                  TIMESTAMP := "TS0",
                  SD_1 := #ME.Pr.N1,
                  SD_2 := #ME.Pr.N2,
                  SD_6 := #ME.Pr.N6);
       END_IF;
       // Действие Km1 заблокировано (Ds1/DsA)
       IF (#Mp.Ds1) THEN
           // Сохраняем флаги исполнения
           #ME.Pr.N2.%X2 := #MF.Md.Ds1;
           #ME.Pr.N2.%X1 := #MF.Rn.Ds1;
           #ME.Pr.N2.%X0 := #MF.Ms.Ds1;
           #ME.Pr.N6 := #GRP + #MF.D1;
           // Вызываем ALARM для активных изменений
           #MsDs1(SIG := #Mx.Ds1,
                  TIMESTAMP := "TS0",
                  SD_1 := #ME.Pr.N1,
                  SD_2 := #ME.Pr.N2,
                  SD_6 := #ME.Pr.N6);
       END_IF;
       // Действие Km2 заблокировано (Ds2/DsA)
       IF (#Mp.Ds2) THEN
           // Сохраняем флаги исполнения
           #ME.Pr.N2.%X2 := #MF.Md.Ds2;
           #ME.Pr.N2.%X1 := #MF.Rn.Ds2;
           #ME.Pr.N2.%X0 := #MF.Ms.Ds2;
           #ME.Pr.N6 := #GRP + #MF.D2;
           // Вызываем ALARM для активных изменений
           #MsDs2(SIG := #Mx.Ds2,
                  TIMESTAMP := "TS0",
                  SD_1 := #ME.Pr.N1,
                  SD_2 := #ME.Pr.N2,
                  SD_6 := #ME.Pr.N6);
       END_IF;
       // Отключен автоматический выключатель
       IF (#Mp.QFe) THEN
           // Сохраняем флаги исполнения
           #ME.Pr.N2.%X2 := #MF.Md.QFe;
           #ME.Pr.N2.%X1 := #MF.Rn.QFe;
           #ME.Pr.N2.%X0 := #MF.Ms.QFe;
           #ME.Pr.N6 := #GRP + 12;
           // Вызываем ALARM для активных изменений
           #MsQFe(SIG := #Mx.QFe,
                  TIMESTAMP := "TS0",
                  SD_1 := #ME.Pr.N1,
                  SD_2 := #ME.Pr.N2,
                  SD_6 := #ME.Pr.N6);
       END_IF;
       // Внешняя неисправность (блокирующая)
       IF (#Mp.Flt) THEN
           // Сохраняем флаги исполнения
           #ME.Pr.N2.%X2 := #MF.Md.Flt;
           #ME.Pr.N2.%X1 := #MF.Rn.Flt;
           #ME.Pr.N2.%X0 := #MF.Ms.Flt;
           #ME.Pr.N6 := #GRP + 13;
           // Вызываем ALARM для активных изменений
           #MsFlt(SIG := #Mx.Flt,
                  TIMESTAMP := "TS0",
                  SD_1 := #ME.Pr.N1,
                  SD_2 := #ME.Pr.N2,
                  SD_6 := #ME.Pr.N6);
       END_IF;
       // Внутренняя неисправность DrvCell
       IF (#Mp.Err) THEN
           // Сохраняем флаги исполнения
           #ME.Pr.N2.%X2 := #MF.Md.Err;
           #ME.Pr.N2.%X1 := #MF.Rn.Err;
           #ME.Pr.N2.%X0 := #MF.Ms.Err;
           #ME.Pr.N6 := #GRP + 14;
           // Вызываем ALARM для активных изменений
           #MsErr(SIG := #Mx.Err,
                  TIMESTAMP := "TS0",
                  SD_1 := #ME.Pr.N1,
                  SD_2 := #ME.Pr.N2,
                  SD_6 := #ME.Pr.N6);
       END_IF;
       // Сохраняем текущее состояние сообщений
       #MU.Hs := #Hx;
   END_IF;
   // Сохраняем состояние сообщений для контроля Mse
   #MU.Ms := #Hs;

   // Сохраняем флаги сообщений и статуса для HMI
   #ST := #Hs OR #STu;
   // Получаем действующее состояние выходного командного канала
   #Chx := 0;
   #CFx.Act := 1;
   #CFx.Mdx := #Fx.Mdx;
   #STx.STx := DWORD_TO_BYTE(#Hs);
   // Передаем текущую уставку
   IF (#Fx.Mdx) THEN
       // Выбираем SPx для активной команды Cm1/Cm2
       IF (#Fx.Ks1) THEN
           #STx.SPx := #SK1;
       END_IF;
       IF (#Fx.Ks2) THEN
           #STx.SPx := #SK2;
       END_IF;
   ELSE
       // В ручном режиме используем уставку из командного канала
       #STx.SPx := #STk.SPx;
   END_IF;
   // Новое командное слово в Chx
END_FUNCTION_BLOCK

FUNCTION_BLOCK "DrvBus"   // FB22, SCL
TITLE = 'Управление механизмом от кнопок/автоматики с 0-й блокировкой'
{ S7_Optimized_Access := 'FALSE' }
AUTHOR : SAA
FAMILY : xDRIVER
NAME : DrvBus
VERSION : 3.0
   VAR_INPUT
      Ch1 : DWord := 0;   // Слово командного канала №1 для арбитража
      CF1 AT Ch1 : "DrvCF";
      ST1 AT Ch1 : "DrvST";
      Ch2 : DWord := 0;   // Слово командного канала №2 для арбитража
      CF2 AT Ch2 : "DrvCF";
      ST2 AT Ch2 : "DrvST";
      Ln1 : Bool := 1;   // Наличие связи в линии канала №1
      Ln2 : Bool := 1;   // Наличие связи в линии канала №2
   END_VAR
   VAR_OUTPUT
      Chx : DWord := 0;   // Слово командного канала после арбитража
      CFx AT Chx : "DrvCF";
      STx AT Chx : "DrvST";
   END_VAR
   VAR
      Sm1 : "DrvST";   // Слово командного канала №1 для арбитража
      Sm2 : "DrvST";   // Слово командного канала №2 для арбитража
      Dm1 : Struct   // Индивидуальные данные для каналов статические
         CmA : Bool := 0;   // Наличие текущей активной команды
         Brk : Bool := 0;   // Канал заблокирован активной командой
         Lnx : Bool := 0;   // Наличие связи в линии канала
         Cmd : Byte := 0;   // Предыдущая команда и штамп идентификатора команды
      END_STRUCT;
      Dm2 : Struct   // Индивидуальные данные для каналов статические
         CmA : Bool := 0;   // Наличие текущей активной команды
         Brk : Bool := 0;   // Канал заблокирован активной командой
         Lnx : Bool := 0;   // Наличие связи в линии канала
         Cmd : Byte := 0;   // Предыдущая команда и штамп идентификатора команды
      END_STRUCT;
      StB : Struct   // Быстрое преобразование для штампа
         H : Byte := 0;
         L : Byte := 0;
      END_STRUCT;
      StN AT StB : Int;   // Текущий штамп команды в удобной форме
      Brk : Bool := 0;   // Канал заблокирован активной командой
      Brm : Bool := 0;   // Наличие блокировки в предыдущем цикле
      Rep : Bool := 0;   // Требуется перезапуск арбитра в следующем цикле
   END_VAR
   VAR_TEMP
      Dx1 : Struct   // Индивидуальные данные для каналов временные
         EvL : Bool;   // Событие связи канала
         EvC : Bool;   // Событие команды канала
         EvN : Bool;   // Получена новая команда (изменен штамп)
         CAx : Bool;   // Наличие активности канала
      END_STRUCT;
      Dx2 : Struct   // Индивидуальные данные для каналов временные
         EvL : Bool;   // Событие связи канала
         EvC : Bool;   // Событие команды канала
         EvN : Bool;   // Получена новая команда (изменен штамп)
         CAx : Bool;   // Наличие активности канала
      END_STRUCT;
      EvC : Bool;   // Новое состояние команды
      EvN : Bool;   // Новый штамп команды
      EvB : Bool;   // Событие с изменением состояния блокировки
      CmB : Struct   // Быстрое преобразование BYTE2WORD
         H : Byte;
         L : Byte;
      END_STRUCT;
      CmW AT CmB : Word;
   END_VAR
BEGIN
   // Инициализация
   #Dx1.CAx := 0;
   #Dx2.CAx := 0;
   #EvC := 0;
   #EvN := 0;
   #EvB := 0;
   #CmW := 0;
   // Анализ состояния канала №1
   #Dx1.EvL := #Ln1 XOR #Dm1.Lnx;
   #Dx1.EvC := (#Dm1.Cmd <> #ST1.Cmd) & #Ln1;
   #Dx1.EvN := 0;
   // Анализ состояния канала №2
   #Dx2.EvL := #Ln2 XOR #Dm2.Lnx;
   #Dx2.EvC := (#Dm2.Cmd <> #ST2.Cmd) & #Ln2;
   #Dx2.EvN := 0;
   // Обнаружено событие в канале №1
   IF (#Dx1.EvL OR #Dx1.EvC) THEN
       // Фиксируем наличие активной команды
       #Dm1.CmA := (#CF1.Cm2 = 0 & #CF1.Cm0 OR #CF1.Cm1) & #Ln1;
       // Проверяем блокировку канала
       #Dm1.Brk := (#Dm1.Brk OR #Dx1.EvL) & #Dm1.CmA;
       // Проверка получения новой команды
       #CmB.H := #ST1.Cmd;
       #CmB.L := #ST1.Cmd XOR #Dm1.Cmd;
       #Dx1.EvN := NOT (((#CmW & 16#06FF) = 16#0402) OR ((#CmW & 16#07FF) = 16#0001));
       #Dx1.EvC := #Dx1.EvC & (#Dx1.EvN OR #Dm1.Lnx);
       #Dx1.EvN := #Dx1.EvN & #Dx1.EvC;
       // Фиксируем текущее состояние канала
       #Dm1.Lnx := #Ln1;
   END_IF;
   // Обнаружено событие в канале №2
   IF (#Dx2.EvL OR #Dx2.EvC) THEN
       // Фиксируем наличие активной команды
       #Dm2.CmA := (#CF2.Cm2 = 0 & #CF2.Cm0 OR #CF2.Cm1) & #Ln2;
       // Проверяем блокировку канала
       #Dm2.Brk := (#Dm2.Brk OR #Dx2.EvL) & #Dm2.CmA;
       // Проверка получения новой команды
       #CmB.H := #ST2.Cmd;
       #CmB.L := #ST2.Cmd XOR #Dm2.Cmd;
       #Dx2.EvN := NOT (((#CmW & 16#06FF) = 16#0402) OR ((#CmW & 16#07FF) = 16#0001));
       #Dx2.EvC := #Dx2.EvC & (#Dx2.EvN OR #Dm2.Lnx);
       #Dx2.EvN := #Dx2.EvN & #Dx2.EvC;
       // Фиксируем текущее состояние канала
       #Dm2.Lnx := #Ln2;
   END_IF;
   // Проверяем активность каналов №1 и №2
   #Dx1.CAx := #Dx1.EvN OR #Dm1.CmA;
   #Dx2.CAx := #Dx2.EvN OR #Dm2.CmA;
   // Наличие событий
   IF (#Rep OR #Dx1.EvL OR #Dx1.EvC OR #Dx2.EvL OR #Dx2.EvC) THEN
       // Сбрасываем разовые флаги
       #Rep := 0;
       // Фиксируем флаг блокирования канала
       #Brm := #Brk;
       #Brk := #Brk & (#Dx1.CAx OR #Dx2.CAx) OR #Dx1.CAx & #Dx2.CAx OR #Dm1.Brk OR #Dm2.Brk;
       #EvB := #Brk XOR #Brm;
       // Наличие запросов на изменение команды и штампа
       #EvC := #Dx1.EvC OR #Dx2.EvC;
       #EvN := #Dx1.EvN OR #Dx2.EvN;
       // При коротких блокировках повторяем событие
       #Rep := #Brk & #EvN;
       // Выполнение арбитража событий
       IF (#EvB OR (#EvC & NOT #Brk)) THEN
           // Проверка на необходимость изменения штампа
           IF (#EvN OR #Brk) THEN
               #StN := #StN + 8;
           END_IF;
           // Выбор источника текущей команды
           IF (#EvB) THEN
               // Команда СТОП (Активная/Эхо)
               #STx.Cmd := #StB.L;
               #CFx.Cm0 := #Brk;
           ELSE
               // Передаем текущую команду канала №1
               IF (#Dx1.EvC & NOT #Dx2.EvN) THEN
                   #STx.Cmd := #StB.L OR #ST1.Cmd & 16#07;
               END_IF;
               // Передаем текущую команду канала №2
               IF (#Dx2.EvC & NOT #Dx1.EvN) THEN
                   #STx.Cmd := #StB.L OR #ST2.Cmd & 16#07;
               END_IF;
           END_IF;
       END_IF;
   END_IF;
   // Фиксируем текущее состояние каналов
   #Dm1.Cmd := #ST1.Cmd;
   #Dm2.Cmd := #ST2.Cmd;
   // Формируем текущую уставку по последнему активному каналу
   IF (#Dx1.CAx & NOT #Dx2.CAx) THEN
       #STx.SPx := #ST1.SPx;
   END_IF;
   IF (#Dx2.CAx & NOT #Dx1.CAx) THEN
       #STx.SPx := #ST2.SPx;
   END_IF;
   // Формируем статусные флаги после арбитража
   IF (NOT #Ln1) THEN
       // Обнуляем канал при отсутствии связи
       #Ch1 := 0;
       // Устанавливаем флаг сообщения об обрыве связи
       #CF1.MsD := 1;
   END_IF;
   IF (NOT #Ln2) THEN
       // Обнуляем канал при отсутствии связи
       #Ch2 := 0;
       // Устанавливаем флаг сообщения об обрыве связи
       #CF2.MsD := 1;
   END_IF;
   #STx.STx := #ST1.STx OR #ST2.STx;
   #STx.WKx := #ST1.WKx OR #ST2.WKx;
   // Формируем флаг сообщения о блокировке канала
   #CFx.MsB := #CFx.MsB OR #Brk;
   // Результат арбитража каналов в Chx
END_FUNCTION_BLOCK

FUNCTION_BLOCK "DrvSb"   // FB24, SCL
TITLE = 'Управление механизмом от кнопок/автоматики с 0-й блокировкой'
{ S7_Optimized_Access := 'FALSE' }
AUTHOR : SAA
FAMILY : xDRIVER
NAME : DrvSb
VERSION : 3.0
   VAR_INPUT
      Chr : DWord := 0;   // Входное слово командного канала
      CFr AT Chr : "DrvCF";
      STr AT Chr : "DrvST";
      Lnr : Bool := 1;   // Наличие связи в линии командного канала
      SB1 : Bool := 0;   // Кнопка включения Km1 (фронт активен) (с фиксацией или без)
      SB2 : Bool := 0;   // Кнопка включения Km2 (фронт активен) (с фиксацией или без)
      OFF : Bool := 0;   // Кнопка 'СТОП' для снятия фиксации (1==активен)
      Ack : Bool := 0;   // Сброс индикации ошибки (квитирование) (1==активен)
      SBe : Bool := 1;   // Разрешение кнопок (при ==0 запрет без отключения)
      SP1 : SInt := 100;   // Уставка задания Km1 (-100..+100)[%]
      SP2 : SInt := -100;   // Уставка задания Km2 (-100..+100)[%]
      Kb_Sb1 : Bool := 0;   // Кнопка SB1 без фиксации (Km1 отключается после отпускания SB1)
      Kb_Sr1 : Bool := 0;   // Кнопка SB1 в режиме переключателя (Вкл/Откл одной кнопкой)
      Kb_Sb2 : Bool := 0;   // Кнопка SB2 без фиксации (Km2 отключается после отпускания SB2)
      Kb_Sr2 : Bool := 0;   // Кнопка SB2 в режиме переключателя (Вкл/Откл одной кнопкой)
      Kb_Ls1 : Bool := 0;   // Индикация Km1 желтым светом (Lr+Lg)
      Kb_Ls2 : Bool := 0;   // Индикация Km2 желтым светом (Lr+Lg)
      Kb_LsA : Bool := 0;   // Используется общая подсветка на оба канала Km1/Km2
      Kb_LsH : Bool := 0;   // Моноцветная импульсная индикация неисправностей
      Kb_HMI : Bool := 0;   // Кнопки в режиме импульса HMI (сброс после использования)
   END_VAR
   VAR_OUTPUT
      Chx : DWord := 0;   // Слово командного канала после арбитража
      CFx AT Chx : "DrvCF";
      STx AT Chx : "DrvST";
      Lg1 : Bool := 0;   // Индикация действия от SB1 (зеленый)
      Lg2 : Bool := 0;   // Индикация действия от SB2 (зеленый)
      Lr1 : Bool := 0;   // Индикация действия от SB1 (красный)
      Lr2 : Bool := 0;   // Индикация действия от SB2 (красный)
   END_VAR
   VAR
      Bus : "DrvBus";   // Локальный арбитр командного канала
      Ch1 : DWord := 0;   // Локальное слово командного канала
      CF1 AT Ch1 : "DrvCF";
      ST1 AT Ch1 : "DrvST";
      ST0 : "DrvST";   // Локальное слово 'эхо' команды
      SBm : Bool := 0;   // Разрешение кнопок (при ==0 запрет без отключения)
      Drv : Bool := 0;   // Блок используется внутри DrvCell (не проверять Lnx&Act)
      StB : Struct   // Быстрое преобразование для штампа
         H : Byte := 0;
         L : Byte := 0;
      END_STRUCT;
      StN AT StB : Int;   // Текущий штамп команды в удобной форме
      Fm : Struct   // Контрольная структура сохраненного состояния входов
         Res : Byte;   // Резервируем старший байт для удобства записи констант
         SB1 : Bool;   // Кнопка включения Km1 (фронт активен) (с фиксацией или без)
         SB2 : Bool;   // Кнопка включения Km2 (фронт активен) (с фиксацией или без)
         OFF : Bool;   // Кнопка 'СТОП' для снятия фиксации (1==активен)
      END_STRUCT;
      Wm AT Fm : Word;   // Текущее состояние группы входов
   END_VAR
   VAR_TEMP
      Sx1 : Bool;   // События соответствуют нажатию SB1/SB2
      Sx2 : Bool;   // События соответствуют нажатию SB1/SB2
      Lx1 : Bool;   // Наличие события рабочей подсветки (зеленой)
      Lx2 : Bool;   // Наличие события рабочей подсветки (зеленой)
      Tck : Bool;   // Флаг аварийного мигания
      ErA : Bool;   // Флаг аварийного мигания
      Fx : Struct   // Контрольная структура текущего состояния входов
         Res : Byte;   // Резервируем старший байт для удобства записи констант
         SB1 : Bool;   // Кнопка включения Km1 (фронт активен) (с фиксацией или без)
         SB2 : Bool;   // Кнопка включения Km2 (фронт активен) (с фиксацией или без)
         OFF : Bool;   // Кнопка 'СТОП' для снятия фиксации (1==активен)
      END_STRUCT;
      Wx AT Fx : Word;   // Буффер для групповой обработки входов
      Fp : Struct   // Контрольная структура текущего состояния входов
         Res : Byte;   // Резервируем старший байт для удобства записи констант
         SB1 : Bool;   // Кнопка включения Km1 (фронт активен) (с фиксацией или без)
         SB2 : Bool;   // Кнопка включения Km2 (фронт активен) (с фиксацией или без)
         OFF : Bool;   // Кнопка 'СТОП' для снятия фиксации (1==активен)
      END_STRUCT;
      Wp AT Fp : Word;   // Буффер для групповой обработки входов
   END_VAR
BEGIN
   // Инициализируем VAR_TEMP структуру исходным значением
   #Wx := 0;
   #Wp := 0;
   #Sx1 := 0;
   #Sx2 := 0;
   #Lx1 := 0;
   #Lx2 := 0;
   #Tck := 0;
   #ErA := 0;
   // Проверяем текущее эквивалентное состояние входов (с учетом Ключ-Бирки SBe)
   IF (#SBe) THEN
       // Есть разрешение на использование кнопок (от Ключ-Бирки SBe)
       #Fx.SB1 := #SB1;
       #Fx.SB2 := #SB2;
       #Fx.OFF := (#SBm = 0 OR #Fm.OFF) & (#Fx.SB1 OR #Fx.SB2) OR (#Fx.SB1 & #Fx.SB2) OR #OFF;
   END_IF;
   // Проверяем наличие событий
   IF (#Wx <> #Wm) THEN
       // Устанавливаем флаги приходящих событий
       #Wp := #Wx XOR #Wm;
       // Проверяем нажатие/отпускание кнопок
       IF (#Wp = #Wm) THEN
           // Отпущена кнопка или прервана команда
           #ST1.Cmd := #ST0.Cmd;
           // Обнуляем уставку SPx если не SA1/SA2
           IF (NOT #CF1.Cm2) THEN
               #ST1.SPx := 0;
           END_IF;
       ELSE
           // Проверяем на приходящее событие
           #Sx1 := (#Wx = 1) & #Fp.SB1;
           #Sx2 := (#Wx = 2) & #Fp.SB2;
           IF (#Fx.OFF & #Fp.OFF OR #Sx1 OR #Sx2) THEN
               // По умолчанию действие кнопки OFF
               #StN := #StN + 8;
               #ST1.Cmd := #StB.L OR 2#001;
               #ST0.Cmd := #StB.L;
               #ST1.SPx := 0;
               // Действие SB1/SA1
               IF (#Sx1) THEN
                   IF (#Kb_Sb1) THEN
                       // Включение без фиксации SB1
                       #ST1.Cmd := #StB.L OR 2#010;
                   ELSIF (#Kb_Sr1 = 0 OR (#Drv OR #Lnr & #CFr.Act) & #CFr.Ks1 = 0) THEN
                       // Включение с фиксацией SA1
                       #ST1.Cmd := #StB.L OR 2#110;
                       #ST0.Cmd := #StB.L OR 2#100;
                   END_IF;
               END_IF;
               // Действие SB2/SA2
               IF (#Sx2) THEN
                   IF (#Kb_Sb2) THEN
                       // Включение без фиксации SB2
                       #ST1.Cmd := #StB.L OR 2#011;
                   ELSIF (#Kb_Sr2 = 0 OR (#Drv OR #Lnr & #CFr.Act) & #CFr.Ks2 = 0) THEN
                       // Включение с фиксацией SA1
                       #ST1.Cmd := #StB.L OR 2#111;
                       #ST0.Cmd := #StB.L OR 2#101;
                   END_IF;
               END_IF;
           END_IF;
       END_IF;
       // Сохраняем текущее состояние входов
       #Wm := #Wx;
   END_IF;
   // Передаем текущую уставку при работе в режиме джойстика
   IF (#CF1.Cm1) THEN
       // Выбираем SPx для активной команды SA1/SB1/SA2/SB2
       IF (#CF1.Cm0) THEN
           #ST1.SPx := #SP2;
       ELSE
           #ST1.SPx := #SP1;
       END_IF;
   END_IF;
   // Фиксируем текущее состояние Ключ-Бирки
   #SBm := #SBe;
   // Фиксируем сигнал квитирования
   #CF1.Ack := #Ack & #SBe;
   // Проводим сброс входов в режиме HMI
   IF (#Kb_HMI) THEN
       #SB1 := 0;
       #SB2 := 0;
       #OFF := 0;
       #Ack := 0;
   END_IF;
   // Формируем ST1.STx при использовании в DrvCell
   IF (#Drv) THEN
       #ST1.STx := #STr.STx;
       #CF1.Act := 1;
   END_IF;
   // Вызов блока арбитра и выдача командного канала
   #Bus(Ch1 := #Ch1,
        Ch2 := #Chr,
        Ln1 := 1,
        Ln2 := #Lnr,
        Chx => #Chx);
   // Иллюминация с возможностью вывода на PP17
   #Tck := "_Clk08sec" & "_Clk04sec" & "_Clk02sec" & #Kb_LsH;
   #Lx1 := (#CFx.Ks1 & "_Clk08sec" OR #CFx.Tm1 OR #CFx.Sx1) & #CFx.Er1 = 0;
   #Lx2 := (#CFx.Ks2 & "_Clk08sec" OR #CFx.Tm2 OR #CFx.Sx2) & #CFx.Er2 = 0;
   IF (#Kb_LsA) THEN
       // Выводим на общий индикатор
       #ErA := #CFx.Er1 OR #CFx.Er2;
       #Lg1 := (#Lx1 OR #Lx2) & #ErA = 0 OR #ErA & #Tck;
       #Lr1 := #ErA OR #Lx1 & #Kb_Ls1 OR #Lx2 & #Kb_Ls2;
       #Lg2 := 0;
       #Lr2 := 0;
   ELSE
       // Раздельная индикация каналов
       #Lg1 := #Lx1 OR #CFx.Er1 & #Tck;
       #Lg2 := #Lx2 OR #CFx.Er2 & #Tck;
       #Lr1 := #CFx.Er1 OR #Lx1 & #Kb_Ls1;
       #Lr2 := #CFx.Er2 OR #Lx2 & #Kb_Ls2;
   END_IF;
   // Результат арбитража каналов в Chx
END_FUNCTION_BLOCK

FUNCTION_BLOCK "AiMd"   // FB32, SCL
TITLE = 'Настройка входного аналогового канала'
{ S7_Optimized_Access := 'FALSE' }
AUTHOR : SAA
FAMILY : xSENSOR
NAME : AiMd
VERSION : 4.0
   VAR_INPUT
      Md_Nm : Bool := 0;   // Pn указывает нормальный==0/номинальный==1 сигнал
      Md_Ke : Bool := 0;   // Прямое использование Kf и Zp (с перерассчетом P1 и P0)
      Md_Ms : Bool := 1;   // Разрешена генерация сообщений и использование Pn
      Md_Rt : Bool := 0;   // Круговой датчик с переходом через 0 (однооборотный/многооборотный)
      Md_Rh : Bool := 1;   // Для кругового датчика использовать шкалу со знаком (-180*..+180*)
      Md_An : DInt := DINT#27648;   // Значение PIW/PID(Ai/Ad) при 100% входного диапазона
      Md_P1 : Real := 100.0;   // Номинал Px при Ai=100% (Ai=An[1]) [E]
      Md_P0 : Real := 0.0;   // Номинал Px при Ai=0% (Ai=0[1]) [E]
      Md_Kf : Real := 1.0;   // Коэффициент преобразования Ai=>Px (множитель) [E/1]
      Md_Kx : Real := 1.0;   // Множитель для сглаживания колебаний входного сигнала
      Md_dP : Real := 0.0;   // Гистерезис в определении уровней
      Md_Pn : Real := 1.0e+38;   // Номинальный/Нормальный уровень сигнала [E]
      Md_Ha : Real := 1.0e+38;   // Верхний уровень сигнала: Аварийный [E/%]
      Md_La : Real := -1.0e+38;   // Нижний уровень сигнала: Аварийный [E/%]
      Md_Hw : Real := 1.0e+38;   // Верхний уровень сигнала: Предупредительный [E/%]
      Md_Lw : Real := -1.0e+38;   // Нижний уровень сигнала: Предупредительный [E/%]
      Md_H1 : Real := 1.0e+38;   // Верхний уровень сигнала: Рабочая зона 1 [E/%]
      Md_L1 : Real := -1.0e+38;   // Нижний уровень сигнала: Рабочая зона 1 [E/%]
      Md_H0 : Real := 1.0e+38;   // Верхний уровень сигнала: Рабочая зона 0 [E/%]
      Md_L0 : Real := -1.0e+38;   // Нижний уровень сигнала: Рабочая зона 0 [E/%]
   END_VAR
   VAR_OUTPUT
      Ch : "AiSP";   // Заданные настройки входного аналогового канала
   END_VAR
BEGIN
   // Производится настройка аналогового канала
   #Ch."M".Nm := #Md_Nm;
   #Ch."M".Ke := #Md_Ke;
   #Ch."M".Ms := #Md_Ms;
   #Ch."M".Rt := #Md_Rt;
   #Ch."M".Rh := #Md_Rh;
   #Ch."M".An := #Md_An;
   #Ch."M".P1 := #Md_P1;
   #Ch."M".P0 := #Md_P0;
   #Ch."M".Kf := #Md_Kf;
   #Ch."M".Kx := #Md_Kx;
   #Ch."M".dP := #Md_dP;
   #Ch.Pn := #Md_Pn;
   #Ch.Ha := #Md_Ha;
   #Ch.La := #Md_La;
   #Ch.Hw := #Md_Hw;
   #Ch.Lw := #Md_Lw;
   #Ch.H1 := #Md_H1;
   #Ch.L1 := #Md_L1;
   #Ch.H0 := #Md_H0;
   #Ch.L0 := #Md_L0;
   // Проверяем непротиворечивость данных
   IF (#Ch."M".Nm & #Ch.Pn = 0.0) THEN
       #Ch.Pn := 100.0;
   END_IF;
   IF (#Ch."M".An = 0) THEN
       #Ch."M".An := 27648;
   END_IF;
   // Формируем набор коэффициентов
   IF (#Ch."M".Ke) THEN
       #Ch."M".P1 := #Ch."M".P0 + DINT_TO_REAL(#Ch."M".An) * #Ch."M".Kf;
   ELSE
       #Ch."M".Kf := (#Ch."M".P1 - #Ch."M".P0) / DINT_TO_REAL(#Ch."M".An);
   END_IF;
   // Сохраняем признак изменения настройки
   #Ch."M".Rz := 1;
   #Ch."M".Rs := 0;
   // Настройки сохранены в Ch
END_FUNCTION_BLOCK

FUNCTION_BLOCK "AiCh"   // FB33, SCL
TITLE = 'Обработка входного аналогового канала'
{ S7_Optimized_Access := 'FALSE' }
AUTHOR : SAA
FAMILY : xSENSOR
NAME : AiCh
VERSION : 5.0
// Блок используется для обработки аналоговых и цифровых датчиков,
// т.е. для обработки каналов модулей аналогового ввода, модулей
// обработки датчиков SSI и датчиков с интерфейсом PROFIBUS.
// Настройка диапазона производится общим каналом для однотипных
// датчиков. Предполагается контроль нескольких уровней сигнала
// с возможностью выдачи сообщений.
   VAR_INPUT
      GRP : UDInt := 0;   // Группа механизмов для HMI
      CW : DWord := 0;   // Текущее слово управления от HMI
      CF AT CW : "AiSF";   // Побитная расшифровка слова управления
      Ai : Int := 0;   // Текущее значение аналогового входного канала [1]
      Pr : DWord := 16#00000000;   // Текущее значение цифрового канала датчика [1]
      Ph : Real := 0.0;   // Заданное значение плавающего смещения канала [E]
      SF : Real := 0.0;   // Заданное значение канала (для форсирования) [E]
      SP : Real := 0.0;   // Заданное положение датчика (для настройки) [E]
      SPn : Real := 1.0e+38;   // Номинальный/Нормальный уровень сигнала [E]
      SHa : Real := 1.0e+38;   // Верхний уровень сигнала: Аварийный [E/%]
      SLa : Real := -1.0e+38;   // Нижний уровень сигнала: Аварийный [E/%]
      SHw : Real := 1.0e+38;   // Верхний уровень сигнала: Предупредительный [E/%]
      SLw : Real := -1.0e+38;   // Нижний уровень сигнала: Предупредительный [E/%]
      SH1 : Real := 1.0e+38;   // Верхний уровень сигнала: Рабочая зона 1 [E/%]
      SL1 : Real := -1.0e+38;   // Нижний уровень сигнала: Рабочая зона 1 [E/%]
      SH0 : Real := 1.0e+38;   // Верхний уровень сигнала: Рабочая зона 0 [E/%]
      SL0 : Real := -1.0e+38;   // Нижний уровень сигнала: Рабочая зона 0 [E/%]
      LFQ : Bool := 0;   // Запрос режима форсирования (PLC)
      LSP : Bool := 0;   // Запрос установки смещения (PLC)
      HWx : Bool := 0;   // Дополнительная сигнализация на HMI
      HWa : Bool := 0;   // Дополнительная сигнализация на HMI (авария)
      MEn : Bool := 1;   // Разрешение выдачи сообщений для HMI
      Md_MFt : Bool := 1;   // Разрешено сообщение Err (Неисправность канала датчика)
      Md_MHa : Bool := 1;   // Разрешено сообщение QHa (Верхний уровень сигнала: Аварийный)
      Md_MLa : Bool := 1;   // Разрешено сообщение QLa (Нижний уровень сигнала: Аварийный)
      Md_MHw : Bool := 1;   // Разрешено сообщение QHw (Верхний уровень сигнала: Предупредительный)
      Md_MLw : Bool := 1;   // Разрешено сообщение QLw (Нижний уровень сигнала: Предупредительный)
      Md_MH1 : Bool := 0;   // Разрешено сообщение QH1 (Верхний уровень сигнала: Рабочая зона 1)
      Md_ML1 : Bool := 0;   // Разрешено сообщение QL1 (Нижний уровень сигнала: Рабочая зона 1)
      Md_MH0 : Bool := 0;   // Разрешено сообщение QH0 (Верхний уровень сигнала: Рабочая зона 0)
      Md_ML0 : Bool := 0;   // Разрешено сообщение QL0 (Нижний уровень сигнала: Рабочая зона 0)
      Md_HHa : Bool := 1;   // Наличие сигнала QHa==1 отображать в SW как аварию
      Md_HLa : Bool := 1;   // Наличие сигнала QLa==1 отображать в SW как аварию
      Md_HHw : Bool := 0;   // Наличие сигнала QHw==1 отображать в SW как аварию
      Md_HLw : Bool := 0;   // Наличие сигнала QLw==1 отображать в SW как аварию
      Md_EFQ : Bool := 1;   // Разрешение форсирования (HMI)
      Md_ESP : Bool := 1;   // Разрешение установки смещения (HMI)
      Md_EPx : Bool := 0;   // Разрешение принудительного значения при неисправности канала
      Md_FPx : Real := 0.0;   // Принудительно задаваемое значение при неисправности канала
      Md_KPx : Real := 1.0;   // Поправочный коэффициент (для зеркальной установки датчика -1.0)
      Md_LPr : DWord := 16#01FFFFFF;   // Маска значащих битов данных в Pr
      Md_FPr : DWord := 16#30000000;   // Маска флагов неисправности в Pr
      Ch : "AiSP";   // Заданные настройки входного аналогового канала
   END_VAR
   VAR_OUTPUT
      NDB : UDInt := 0;   // Номер InstanceDB
      SW : DWord := 0;   // Текущее слово состояния для HMI
      Pw : DInt := 0;   // Текущее фактическое состояние канала [1]
      Pz : Real := 0.0;   // Текущее фактическое состояние канала [E]
      Px : Real := 0.0;   // Текущее рабочее состояние канала [E]
      QFt : Bool := 0;   // Неисправность канала датчика
      QHa : Bool := 0;   // Верхний уровень сигнала: Аварийный
      QLa : Bool := 0;   // Нижний уровень сигнала: Аварийный
      QHw : Bool := 0;   // Верхний уровень сигнала: Предупредительный
      QLw : Bool := 0;   // Нижний уровень сигнала: Предупредительный
      QH1 : Bool := 0;   // Верхний уровень сигнала: Рабочая зона 1
      QL1 : Bool := 0;   // Нижний уровень сигнала: Рабочая зона 1
      QH0 : Bool := 0;   // Верхний уровень сигнала: Рабочая зона 0
      QL0 : Bool := 0;   // Нижний уровень сигнала: Рабочая зона 0
   END_VAR
   VAR_IN_OUT
      ZP : Real := 0.0;   // Смещение нуля датчика (для сохранения) [E]
   END_VAR
   VAR
      MsQFt : Program_Alarm;   // Неисправность канала датчика
      MsQHa : Program_Alarm;   // Верхний уровень сигнала: Аварийный
      MsQLa : Program_Alarm;   // Нижний уровень сигнала: Аварийный
      MsQHw : Program_Alarm;   // Верхний уровень сигнала: Предупредительный
      MsQLw : Program_Alarm;   // Нижний уровень сигнала: Предупредительный
      MsQH1 : Program_Alarm;   // Верхний уровень сигнала: Рабочая зона 1
      MsQL1 : Program_Alarm;   // Нижний уровень сигнала: Рабочая зона 1
      MsQH0 : Program_Alarm;   // Верхний уровень сигнала: Рабочая зона 0
      MsQL0 : Program_Alarm;   // Нижний уровень сигнала: Рабочая зона 0
      ST : "AiSF";   // Буффер флагов состояния канала
      ME : "DrvME";   // Набор данных для обработки ALARM_D
   END_VAR
   VAR_TEMP
      TSA : "TANY";   // Структура ANY для определения InstanceDB
      TPA AT TSA : ANY;   // Указатель ANY для определения InstanceDB
      Fx : "AiSF";   // Побитная расшифровка слова состояния
      Dx AT Fx : DWord;   // Буффер для текущих флагов
      Fm : "AiSF";   // Побитная расшифровка слова состояния
      Dm AT Fm : DWord;   // Буффер для сохраненных флагов
      Fp : "AiSF";   // Побитная расшифровка слова состояния
      Dp AT Fp : DWord;   // Буффер для признаков изменения флагов
      PxN : Real;   // Px с учетом гистерезиса Cz.M.dP и номинала SPn
      PxH : Real;   // Px с учетом гистерезиса Cz.M.dP и номинала SPn
      PxL : Real;   // Px с учетом гистерезиса Cz.M.dP и номинала SPn
      Pu : Real;   // Локальное значение (для рассчетов)
      Pv : DInt;   // Локальное значение (для рассчетов)
      Pd : DWord;   // Локальное значение (для рассчетов)
      Fz : Bool;   // Признак наличия сообщения
   END_VAR
BEGIN
   // Загружаем текущие флаги состояния
   #Fm := #ST;
   #Fx := #ST;
   // Фиксируем запрос на параметризацию
   IF (#Ch."M".Rs XOR #Ch."M".Rz) THEN
       #Ch."M".Rs := #Ch."M".Rz;
       #Ch."M".Kf := #Ch."M".Kf * #Md_KPx;
       #SPn := #Ch.Pn;
       #SHa := #Ch.Ha;
       #SLa := #Ch.La;
       #SHw := #Ch.Hw;
       #SLw := #Ch.Lw;
       #SH1 := #Ch.H1;
       #SL1 := #Ch.L1;
       #SH0 := #Ch.H0;
       #SL0 := #Ch.L0;
       #Fm.QSt := 0;
   END_IF;
   // Фиксируем изменения режима работы
   // Настройка блока выполнена (первый цикл PLC)
   #Fx.QSt := 1;
   // Разрешение выдачи сообщений (HMI)
   #Fx.MEn := #MEn & #Ch."M".Ms & "_MEn";
   // Признак установки смещения
   #Fx.ESP := #Md_ESP;
   #Fx.HSP := #Fx.ESP & #CF.HSP;
   #Fx.LSP := #LSP;
   #Fx.QSP := #Fx.LSP OR #Fx.HSP;
   #CF.HSP := 0;
   // Признак режима форсирования
   #Fx.EFQ := #Md_EFQ;
   #Fx.HFQ := #Fx.EFQ & #CF.HFQ;
   #Fx.LFQ := #LFQ;
   #Fx.QFQ := #Fx.LFQ OR #Fx.HFQ;
   // Наличие неисправности канала
   #Fx.QFt := (INT_TO_WORD(#Ai - 32767) & W#16#FFFE) = 0 OR (#Pr & #Md_FPr) <> 0;
   // Обрабатываем текущие показания канала с учетом типа датчика
   // Фиксируем бинарное значение канала
   #Pw := DWORD_TO_DINT(#Pr & #Md_LPr) + INT_TO_DINT(#Ai);
   // Фиксируем абсолютное значение канала
   #Pz := DINT_TO_REAL(#Pw) * #Ch."M".Kf + #Ch."M".P0;
   // Формируем рабочее значение канала
   IF (#Fx.QFQ) THEN
       // Команда форсирования принудительно устанавливает рабочее значение сигнала
       #Px := #SF;
   ELSIF (#Fx.QFt & #Md_EPx) THEN
       // При неисправности канала (по настройке) используется предустановленное значение
       #Px := #Md_FPx;
   ELSE
       // Фиксируем текущее рабочее значение канала
       #Pu := #Pz - #ZP + #Ph;
       // Для многооборотного датчика производим выравнивание границ
       IF (#Ch."M".Rt) THEN
           // Обрезаем диапазон до размера маски датчика
           #Pv := DWORD_TO_DINT(DINT_TO_DWORD(ROUND(#Pu / ABS(#Ch."M".Kf))) & #Md_LPr);
           IF (#Ch."M".Rh) THEN
               // Формируем знак из старшего бита по маске датчика
               #Pd := (SHR(IN := #Md_LPr, N := 1) XOR #Md_LPr) & #Md_LPr;
               #Pv := DWORD_TO_DINT(DINT_TO_DWORD(#Pv) XOR #Pd) - DWORD_TO_DINT(#Pd);
           END_IF;
           #Pu := DINT_TO_REAL(#Pv) * ABS(#Ch."M".Kf);
       ELSE
           // Производим сглаживание сигнала при необходимости
           #Pu := (#Pu - #Px) * #Ch."M".Kx + #Px;
       END_IF;
       // Сохраняем текущее рабочее значение канала
       #Px := #Pu;
   END_IF;
   // Обработка признака нормального/номинального уровня
   IF (#Ch."M".Nm) THEN
       // Для номинального уровня фиксируем отклонение сигнала [%]
       #PxN := (#Px / #SPn - 1.0) * 100.0;
   ELSE
       // Для нормального уровня фиксируем отклонение сигнала [E]
       #PxN := #Px - #SPn;
   END_IF;
   // Фиксируем TEMP значение сигнала с учетом гистерезиса для компенсации дребезга
   #PxH := #PxN + #Ch."M".dP;
   #PxL := #PxN - #Ch."M".dP;
   // Фиксируем положение виртуальных КВ
   #Fx.QHa := (#Fx.QHa OR (#PxL > #SHa)) & (#PxH > #SHa);
   #Fx.QLa := (#Fx.QLa OR (#PxH < #SLa)) & (#PxL < #SLa);
   #Fx.QHw := (#Fx.QHw OR (#PxL > #SHw)) & (#PxH > #SHw);
   #Fx.QLw := (#Fx.QLw OR (#PxH < #SLw)) & (#PxL < #SLw);
   #Fx.QH1 := (#Fx.QH1 OR (#PxL > #SH1)) & (#PxH > #SH1);
   #Fx.QL1 := (#Fx.QL1 OR (#PxH < #SL1)) & (#PxL < #SL1);
   #Fx.QH0 := (#Fx.QH0 OR (#PxL > #SH0)) & (#PxH > #SH0);
   #Fx.QL0 := (#Fx.QL0 OR (#PxH < #SL0)) & (#PxL < #SL0);
   // Фиксируем групповые признаки
   #Fx.QWg := #Fx.QHw OR #Fx.QLw;
   #Fx.QAm := #Fx.QHa OR #Fx.QLa;
   #Fx.HAm := #HWa OR #Fx.QFt OR (#Fx.QHa & #Md_HHa) OR (#Fx.QLa & #Md_HLa) OR (#Fx.QHw & #Md_HHw) OR (#Fx.QLw & #Md_HLw);
   #Fx.HWg := (#HWx OR #Fx.QWg) & (#Fx.HAm = 0);
   // Фиксируем наличие событий
   #Dp := #Dx XOR #Dm;
   IF (#Dp <> 0) THEN
       // Запрос на инициализацию данных
       IF (#Fp.QSt) THEN
           // Инициализация данных
           #ME.Pr.N2 := 0;
           #ME.Pr.N4 := 0;
           #ME.Pr.N5 := 0;
           // Устанавливаем номер данного Instance Data Block
           #TPA := #ME;
           #NDB := #TSA.PTR.DN;
           // Назначаем группу сообщений (механизмов)
           IF (#GRP = 0) THEN
               #GRP := #NDB * 100;
           END_IF;
       END_IF;
       // Устанавливаем активность сообщений
       // Разрешения MFt/MH*/ML* не проверяются на изменение
       // Сообщение: Неисправность канала датчика
       #Fz := #Fx.QFt & #Md_MFt & #Fx.MEn;
       IF (#Fz XOR #MsQFt.SIG) THEN
           #ME.Pr.N1 := #GRP;
           #ME.Pr.N2.%X0 := #Fm.QFt;
           #ME.Pr.N6 := #GRP + 1;
           #MsQFt(SIG := #Fz,
                  TIMESTAMP := "TS0",
                  SD_1 := #ME.Pr.N1,
                  SD_2 := #ME.Pr.N2,
                  SD_6 := #ME.Pr.N6);
       END_IF;
       // Сообщение: Верхний уровень сигнала: Аварийный
       #Fz := #Fx.QHa & #Md_MHa & #Fx.MEn;
       IF (#Fz XOR #MsQHa.SIG) THEN
           #ME.Pr.N1 := #GRP;
           #ME.Pr.N2.%X0 := #Fm.QHa;
           #ME.Pr.N6 := #GRP + 2;
           #MsQHa(SIG := #Fz,
                  TIMESTAMP := "TS0",
                  SD_1 := #ME.Pr.N1,
                  SD_2 := #ME.Pr.N2,
                  SD_6 := #ME.Pr.N6,
                  SD_7 := #Px,
                  SD_8 := #PxN,
                  SD_9 := #SHa);
       END_IF;
       // Сообщение: Нижний уровень сигнала: Аварийный
       #Fz := #Fx.QLa & #Md_MLa & #Fx.MEn;
       IF (#Fz XOR #MsQLa.SIG) THEN
           #ME.Pr.N1 := #GRP;
           #ME.Pr.N2.%X0 := #Fm.QLa;
           #ME.Pr.N6 := #GRP + 3;
           #MsQLa(SIG := #Fz,
                  TIMESTAMP := "TS0",
                  SD_1 := #ME.Pr.N1,
                  SD_2 := #ME.Pr.N2,
                  SD_6 := #ME.Pr.N6,
                  SD_7 := #Px,
                  SD_8 := #PxN,
                  SD_9 := #SLa);
       END_IF;
       // Сообщение: Верхний уровень сигнала: Предупредительный
       #Fz := #Fx.QHw & #Md_MHw & #Fx.MEn;
       IF (#Fz XOR #MsQHw.SIG) THEN
           #ME.Pr.N1 := #GRP;
           #ME.Pr.N2.%X0 := #Fm.QHw;
           #ME.Pr.N6 := #GRP + 4;
           #MsQHw(SIG := #Fz,
                  TIMESTAMP := "TS0",
                  SD_1 := #ME.Pr.N1,
                  SD_2 := #ME.Pr.N2,
                  SD_6 := #ME.Pr.N6,
                  SD_7 := #Px,
                  SD_8 := #PxN,
                  SD_9 := #SHw);
       END_IF;
       // Сообщение: Нижний уровень сигнала: Предупредительный
       #Fz := #Fx.QLw & #Md_MLw & #Fx.MEn;
       IF (#Fz XOR #MsQLw.SIG) THEN
           #ME.Pr.N1 := #GRP;
           #ME.Pr.N2.%X0 := #Fm.QLw;
           #ME.Pr.N6 := #GRP + 5;
           #MsQLw(SIG := #Fz,
                  TIMESTAMP := "TS0",
                  SD_1 := #ME.Pr.N1,
                  SD_2 := #ME.Pr.N2,
                  SD_6 := #ME.Pr.N6,
                  SD_7 := #Px,
                  SD_8 := #PxN,
                  SD_9 := #SLw);
       END_IF;
       // Сообщение: Верхний уровень сигнала: Рабочая зона 1
       #Fz := #Fx.QH1 & #Md_MH1 & #Fx.MEn;
       IF (#Fz XOR #MsQH1.SIG) THEN
           #ME.Pr.N1 := #GRP;
           #ME.Pr.N2.%X0 := #Fm.QH1;
           #ME.Pr.N6 := #GRP + 6;
           #MsQH1(SIG := #Fz,
                  TIMESTAMP := "TS0",
                  SD_1 := #ME.Pr.N1,
                  SD_2 := #ME.Pr.N2,
                  SD_6 := #ME.Pr.N6,
                  SD_7 := #Px,
                  SD_8 := #PxN,
                  SD_9 := #SH1);
       END_IF;
       // Сообщение: Нижний уровень сигнала: Рабочая зона 1
       #Fz := #Fx.QL1 & #Md_ML1 & #Fx.MEn;
       IF (#Fz XOR #MsQL1.SIG) THEN
           #ME.Pr.N1 := #GRP;
           #ME.Pr.N2.%X0 := #Fm.QL1;
           #ME.Pr.N6 := #GRP + 7;
           #MsQL1(SIG := #Fz,
                  TIMESTAMP := "TS0",
                  SD_1 := #ME.Pr.N1,
                  SD_2 := #ME.Pr.N2,
                  SD_6 := #ME.Pr.N6,
                  SD_7 := #Px,
                  SD_8 := #PxN,
                  SD_9 := #SL1);
       END_IF;
       // Сообщение: Верхний уровень сигнала: Рабочая зона 0
       #Fz := #Fx.QH0 & #Md_MH0 & #Fx.MEn;
       IF (#Fz XOR #MsQH0.SIG) THEN
           #ME.Pr.N1 := #GRP;
           #ME.Pr.N2.%X0 := #Fm.QH0;
           #ME.Pr.N6 := #GRP + 8;
           #MsQH0(SIG := #Fz,
                  TIMESTAMP := "TS0",
                  SD_1 := #ME.Pr.N1,
                  SD_2 := #ME.Pr.N2,
                  SD_6 := #ME.Pr.N6,
                  SD_7 := #Px,
                  SD_8 := #PxN,
                  SD_9 := #SH0);
       END_IF;
       // Сообщение: Нижний уровень сигнала: Рабочая зона 0
       #Fz := #Fx.QL0 & #Md_ML0 & #Fx.MEn;
       IF (#Fz XOR #MsQL0.SIG) THEN
           #ME.Pr.N1 := #GRP;
           #ME.Pr.N2.%X0 := #Fm.QL0;
           #ME.Pr.N6 := #GRP + 9;
           #MsQL0(SIG := #Fz,
                  TIMESTAMP := "TS0",
                  SD_1 := #ME.Pr.N1,
                  SD_2 := #ME.Pr.N2,
                  SD_6 := #ME.Pr.N6,
                  SD_7 := #Px,
                  SD_8 := #PxN,
                  SD_9 := #SL0);
       END_IF;
       // Обработка команды на установку смещения
       IF (#Fx.QSP & #Fp.QSP) THEN
           #ZP := #Pz - #SP + #Ph;
           #Px := #SP;
       END_IF;
       // Сохраняем текущее значение выходов
       #QFt := #Fx.QFt;
       #QHa := #Fx.QHa;
       #QLa := #Fx.QLa;
       #QHw := #Fx.QHw;
       #QLw := #Fx.QLw;
       #QH1 := #Fx.QH1;
       #QL1 := #Fx.QL1;
       #QH0 := #Fx.QH0;
       #QL0 := #Fx.QL0;
       // Сохраняем текущее значение флагов
       #ST := #Fx;
       #SW := #Dx;
   END_IF;
   // Текущее состояние датчика находится в Px/Pz
END_FUNCTION_BLOCK

FUNCTION_BLOCK "MM_T352"   // FB47, SCL
{ S7_Optimized_Access := 'FALSE' }
AUTHOR : AA
FAMILY : xDEVICE
VERSION : 0.1
// Блок моторного модуля SINAMICS (Telegram 352)
   VAR_INPUT
      GRP : UDInt;   // Группа механизмов для HMI
      LA : Hw_Io;   // Адрес периферийной области привода (PI/PQ DEC)
      Vn : Real := 100.0;   // Номинальная скорость [E]
      Vs : Real;   // Заданная скорость [E]
      Ms : Real;   // Заданный момент [%]
      Id : Word;   // Идентификатор дополнительных параметров привода
      DPx : Bool := true;   // Привод управляем (находится в сети DP)
      UBr : Bool;   // Безусловное растормаживание (расжать)
      Enb : Bool := true;   // Разрешение работы (разблокирование)
      KOn : Bool;   // Включить намагничивание V=0 (команда)
      Run : Bool;   // Пуск привода V=Vs (команда)
      Ack : Bool;   // Сброс индикации ошибки (квитирование) (1==активен)
      Mse : Bool := true;   // Разрешение выдачи сообщений для HMI
      Md : Struct
         Ts0 : Time;   // Заданное время отключения намагничивания (KOn|Run)
         EnF : Bool := true;   // Разрешено сообщение Fault (отказ)
         EnA : Bool;   // Разрешено сообщение Alarm (предупреждение)
         Rst : Bool;   // Автоматический перезапуск привода после квитирования
         PZD : Bool;   // Расширенная телеграмма: PZD 10/10
      END_STRUCT;
   END_VAR
   VAR_OUTPUT
      NDB : UDInt := 0;   // Номер InstanceDB
      Re : "DrvRd";   // Данные канала резервирования приводов
      ST : DWord;
      SF AT ST : Struct
         Qm0 : Bool;   // Объект: Устройство ввода резерва
         Qm1 : Bool;   // Объект: Основной привод
         Qm2 : Bool;   // Объект: Резервный привод
         S3 : Bool;
         S4 : Bool;
         S5 : Bool;
         Rd1 : Bool;   // Задейсвован основной ввод
         Rd2 : Bool;   // Задейсвован резервный ввод
         xx : Byte;
         xy : Byte;
         S24 : Bool;
         Alm : Bool;   // Наличие сигнала Alarm (предупреждение)
         Flt : Bool;   // Наличие сигнала Fault (отказ)
         Rdy : Bool;   // Наличие готовности
         S28 : Bool;
         S29 : Bool;
         S30 : Bool;
         S31 : Bool;
      END_STRUCT;
      SW : Word;   // Текущее слово состояния привода
      Vx : Real;   // Текущая скорость привода [E]
      Ix : Real;   // Текущий ток привода [%]
      Mx : Real;   // Текущий момент привода [%]
      An : Int;   // Текущий номер сигнала Alarm [№] (предупреждение) (либо альтернативные данные)
      Fn : Int;   // Текущий номер сигнала Fault [№] (отказ)
      P7 : Int;   // Текущее значение PZD7 [INT] (расширенная телеграмма)
      P8 : Int;   // Текущее значение PZD8 [INT] (расширенная телеграмма)
      P9 : DInt;   // Текущее значение PZD9+PZD10 [DINT] (расширенная телеграмма)
      Rd1 : Bool;   // Данный привод включен как основной
      Rd2 : Bool;   // Данный привод включен как резервный
      Brk : Bool;   // Привод включен (разблокировка тормоза)
      Rdy : Bool;   // Готовность привода к включению
      Flt : Bool;   // Наличие сигнала Fault (отказ)
      Alm : Bool;   // Наличие сигнала Alarm (предупреждение)
      RRD : Int;   // Код выполнения функции чтения данных DPRD_DAT
      RWR : Int;   // Код выполнения функции записи данных DPWR_DAT
      RAD : Int;   // Код выполнения функции S7-сообщений ALARM_D
   END_VAR
   VAR
      MsAlm : Program_Alarm;   // Моторный модуль выдал сигнал предупреждения
      MsFlt : Program_Alarm;   // Модуль управления выдал сигнал аварии
      iT352 : Struct   // Telegram 352 Drive Unit
         PZD1 : Struct
            b08 : Bool;   // 1 = Speed setpoint - actual value deviation within tolerance t_off
            b09 : Bool;   // 1 = Control requested
            b10 : Bool;   // 1 = f or n comparison value reached/exceeded
            b11 : Bool;   // 1 = I, M, or P limit reached
            b12 : Bool;   // 1 = Open the holding brake
            b13 : Bool;   // 1 = No motor overtemperature alarm
            b14 : Bool;   // 1 = Motor rotates forwards (n_act >=0) 0 = Motor rotates backwards (n_act < 0)
            b15 : Bool;   // 1 = No alarm, thermal overload, power unit
            b00 : Bool;   // 1 = Ready for switching on
            b01 : Bool;   // 1 = Ready for operation
            b02 : Bool;   // 1 = Operation enabled
            b03 : Bool;   // 1 = Fault present
            b04 : Bool;   // 1 = No coast down active (OFF2 inactive)
            b05 : Bool;   // 1 = No fast stop active (OFF3 inactive)
            b06 : Bool;   // 1 = Switching on inhibited active
            b07 : Bool;   // 1 = Alarm present
         END_STRUCT;
         PZD2 : Int;   // Текущая скорость привода [%w] (Vr)
         PZD3 : Int;   // Текущий ток привода [%w] (Ir)
         PZD4 : Int;   // Текущий момент привода [%w] (Mr)
         PZD5 : Int;   // Текущее сообщение Alarm [№] (Wx)
         PZD6 : Int;   // Текущее сообщение Fault [№] (Ax)
         PZD7 : Int;   // ----
         PZD8 : Int;
         PZD9 : DInt;
      END_STRUCT;
      iP6 AT iT352 : Struct   // Telegram 352 Drive Unit
         PZD1 : Int;
         PZD2 : Int;
         PZD3 : Int;
         PZD4 : Int;
         PZD5 : Int;
         PZD6 : Int;
      END_STRUCT;
      SWx AT iT352 : Word;   // Текущее слово состояния
      qT352 : Struct   // Telegram 352 Drive Unit
         PZD1 : Struct   // STW1
            b08 : Bool;
            b09 : Bool;
            b10 : Bool := true;   // 1 = Control via PLC
            b11 : Bool;   // 1 = Direction reversal
            b12 : Bool;   // 1 = Unconditionally open the holding brake
            b13 : Bool;   // 1 = Motorized potentiometer setpoint raise
            b14 : Bool;   // 1 = Motorized potentiometer setpoint lower
            b15 : Bool;
            b00 : Bool;   // 1 = ON (pulses can be enabled) 0 = OFF1 (braking with ramp-function generator, then pulse suppression & ready for switching on)
            b01 : Bool := true;   // 1 = No OFF2 (enable is possible) 0 = OFF2 (immediate pulse suppression and switching on inhibited)
            b02 : Bool;   // 1 = No OFF3 (enable possible) 0 = OFF3 (braking with the OFF3 ramp p1135, then pulse suppression and switching on inhibited)
            b03 : Bool := true;   // 1 = Enable operation (pulses can be enabled) 0 = Inhibit operation (suppress pulses)
            b04 : Bool := true;   // 1 = Operating condition (the ramp-function generator can be enabled) 0 = Inhibit ramp-function generator (set the ramp-function generator output to zero)
            b05 : Bool := true;   // 1 = Enable the ramp-function generator 0 = Stop the ramp-function generator (freeze the ramp-function generator output)
            b06 : Bool := true;   // 1 = Enable setpoint 0 = Inhibit setpoint (set the ramp-function generator input to zero)
            b07 : Bool;   // 0 = Acknowledge faults
         END_STRUCT;
         PZD2 : Int;   // Уставка скорости привода [%w] (Vw)
         PZD3 : Int;   // Уставка момента привода [%w] (Mw)
         PZD4 : Word;   // Идентификатор параметров привода (Id)
         PZD5 : Word;
         PZD6 : Word;
         PZD7 : Int;
         PZD8 : Int;
         PZD9 : DInt;
      END_STRUCT;
      qP6 AT qT352 : Struct   // Telegram 352 Drive Unit
         PZD1 : Int;
         PZD2 : Int;
         PZD3 : Int;
         PZD4 : Int;
         PZD5 : Int;
         PZD6 : Int;
      END_STRUCT;
      CWx AT qT352 : Word;   // Текущее слово управления
      Tm1 : Time;   // Время ожидания готовности (Rdy)
      Tm0 : Time;   // Время отключения намагничивания (KOn|Run)
      Bm : DWord := 16#1;   // Буффер флагов состояния привода
      B0 : DWord;   // Буффер вспомогательных данных
      B1 : DWord;   // Буффер вспомогательных данных
      FSc : Bool := 1;   // Первый проход блока (необходима инициализация)
      ME : "DrvME";
   END_VAR
   VAR_TEMP
      TSA : "TANY";   // Структура ANY для определения InstanceDB
      TPA AT TSA : ANY;   // Указатель ANY для определения InstanceDB
      Fx : Struct   // Флаги состояния привода
         w00 : Int;
         Mse : Bool;   // Разрешение выдачи сообщений для HMI
         EnF : Bool;   // Разрешено сообщение Fault (отказ)
         EnA : Bool;   // Разрешено сообщение Alarm (предупреждение)
         MsF : Bool;   // Наличие сообщения Fault (отказ)
         MsA : Bool;   // Наличие сообщения Alarm (предупреждение)
         r25 : Bool;
         r26 : Bool;
         r27 : Bool;
         Res : Bool;   // Первый запуск блока
         Flt : Bool;   // Наличие сигнала Fault (отказ)
         Alm : Bool;   // Наличие сигнала Alarm (предупреждение)
         Rdy : Bool;   // Сигнал готовности привода (b00)
         KOn : Bool;   // Включить привод KOn|Run (команда)
         Run : Bool;   // Наличие результирующей команды на включение привода
         Tx1 : Bool;   // Таймер ожидания готовности (Rdy)
         Tx0 : Bool;   // Таймер паузы отключения намагничивания (KOn|Run)
      END_STRUCT;
      Dx AT Fx : DWord;   // Буффер для текущих флагов
      Fm : Struct
         w00 : Int;
         Mse : Bool;   // Разрешение выдачи сообщений для HMI
         EnF : Bool;   // Разрешено сообщение Fault (отказ)
         EnA : Bool;   // Разрешено сообщение Alarm (предупреждение)
         MsF : Bool;   // Наличие сообщения Fault (отказ)
         MsA : Bool;   // Наличие сообщения Alarm (предупреждение)
         r25 : Bool;
         r26 : Bool;
         r27 : Bool;
         Res : Bool;   // Первый запуск блока
         Flt : Bool;   // Наличие сигнала Fault (отказ)
         Alm : Bool;   // Наличие сигнала Alarm (предупреждение)
         Rdy : Bool;   // Сигнал готовности привода (b00)
         KOn : Bool;   // Включить привод KOn|Run (команда)
         Run : Bool;   // Наличие результирующей команды на включение привода
         Tx1 : Bool;   // Таймер ожидания готовности (Rdy)
         Tx0 : Bool;   // Таймер паузы отключения намагничивания (KOn|Run)
      END_STRUCT;
      dm AT Fm : DWord;   // Буффер для сохраненных флагов
      Fp : Struct
         w00 : Int;
         Mse : Bool;   // Разрешение выдачи сообщений для HMI
         EnF : Bool;   // Разрешено сообщение Fault (отказ)
         EnA : Bool;   // Разрешено сообщение Alarm (предупреждение)
         MsF : Bool;   // Наличие сообщения Fault (отказ)
         MsA : Bool;   // Наличие сообщения Alarm (предупреждение)
         r25 : Bool;
         r26 : Bool;
         r27 : Bool;
         Res : Bool;   // Первый запуск блока
         Flt : Bool;   // Наличие сигнала Fault (отказ)
         Alm : Bool;   // Наличие сигнала Alarm (предупреждение)
         Rdy : Bool;   // Сигнал готовности привода (b00)
         KOn : Bool;   // Включить привод KOn|Run (команда)
         Run : Bool;   // Наличие результирующей команды на включение привода
         Tx1 : Bool;   // Таймер ожидания готовности (Rdy)
         Tx0 : Bool;   // Таймер паузы отключения намагничивания (KOn|Run)
      END_STRUCT;
      Dp AT Fp : DWord;   // Буффер для признаков изменения флагов
      Vm : Real;   // Ограничение уставки скорости
   END_VAR
   VAR CONSTANT
      Ts1 : Time := T#200ms;   // // Заданное время ожидания готовности (Rdy)
   END_VAR
BEGIN
   //=======================================
   // Блок моторного модуля SINAMICS (Telegram 352)
   //
   // Для диагностики используется состояние полученное по сети DP.
   // Управление производится по каналу циклического обмена сети DP.
   // Моторный модуль:
   // (Telegram 352)           PZD 6/6 или
   // (Telegram 352 -> 999)    PZD 10/10
   // Rd PZD1: ZSW1            слово: состояние
   // Rd PZD2: NIST_A_GLATT    слово: текущая скорость, сглаженная
   // Rd PZD3: IAIST_GLATT     слово: текущий ток (модуль), сглаженный
   // Rd PZD4: MIST_GLATT      слово: текущий момент, сглаженный
   // Rd PZD5: WARN_CODE       слово: код предупреждения
   // Rd PZD6: FAULT_CODE      слово: код неисправности
   // Rd PZD7: <Reserved>      слово: ----
   // Rd PZD8: <Reserved>      слово: ----
   // Rd PZD9: RotorHi         слово: старшее слово положения ротора [DINT] (r0094)
   // Rd PZD10:RotorLo         слово: младшее слово положения ротора [DINT] (r0094)
   // Wr PZD1: STW1            слово: управление
   // Wr PZD2: NSOLL_A         слово: заданная скорость
   // Wr PZD3: <Mw>            слово: <заданный момент, опционно>
   // Wr PZD4: <Id>            слово: <заданный параметр, опционно>
   // Wr PZD5: <Reserved>      слово: ----
   // Wr PZD6: <Reserved>      слово: ----
   // Wr PZD7: <Reserved>      слово: ----
   // Wr PZD8: <Reserved>      слово: ----
   // Wr PZD9: <Reserved>      слово: ----
   // Wr PZD10:<Reserved>      слово: ----
   //


